// TwinCAT 3 PLC project PLC_MOTION
// Title: PLC_MOTION_LAYER
// Author: D. Hauer
// ProjectVersion: 01.01.00
// Description: MC-PtP, NCI, Camming cyclic execution layer for motion commands
// ProgramVersion: 3.1.4026.26
// CompilerDefines: TEST, NCI, CAM, XFC
// libraries:
//   Tc2_EtherCAT, * (Beckhoff Automation GmbH)
//   Tc2_MC2, * (Beckhoff Automation GmbH)
//   Tc2_MC2_Camming, * (Beckhoff Automation GmbH)
//   Tc2_MC2_Drive, * (Beckhoff Automation GmbH)
//   Tc2_MC2_FlyingSaw, * (Beckhoff Automation GmbH)
//   Tc2_MC2_XFC, * (Beckhoff Automation GmbH)
//   Tc2_NCI, * (Beckhoff Automation GmbH)
//   Tc2_PlcInterpolation, * (Beckhoff Automation GmbH)
//   Tc2_Standard, * (Beckhoff Automation GmbH)
//   Tc2_System, * (Beckhoff Automation GmbH)
//   Tc2_Utilities, * (Beckhoff Automation GmbH)
//   Tc3_Module, * (Beckhoff Automation GmbH)
// project tree:
//   APPLICATION/ GVL_APPLICATION.TcGVL (not stored)
//   APPLICATION/_types/Application/ E_APP_CHECK.TcDUT, E_APP_VARIANT.TcDUT (not stored), ST_APP_CTRL.TcDUT, ST_APP_STATE.TcDUT (not stored)
//   APPLICATION/_types/LinkedList/ E_LIST_CHECK.TcDUT, E_LIST_CTRL.TcDUT, E_LIST_STATE.TcDUT (not stored), fb_Process_LinkedList.TcPOU, fb_Process_LinkedListCtrl.TcPOU (not stored), I_Process_LinkedList.TcIO, ST_LIST_CTRL.TcDUT (not stored), ST_LIST_NODE_DATA.TcDUT (not stored), ST_LIST_STATE.TcDUT, ST_PROCESS_DATA.TcDUT (not stored), ST_PROCESS_LIST_RESULT.TcDUT
//   MAPPING/ MAPPING_AXIS_in.TcPOU, MAPPING_AXIS_out.TcPOU (not stored)
//   MAPPING/types/ U_AXIS_CTRL.TcDUT (not stored), U_AXIS_NC_PARAMETER_WRT.TcDUT, U_AXIS_HOMING.TcDUT (not stored), U_AXIS_MOTION_OPTIONS.TcDUT, U_AXIS_MOVE_DATA.TcDUT, U_AXIS_GEAR_IN.TcDUT (not stored), U_AXIS_NC_PARAMETER_RD.TcDUT, U_AXIS_STATE.TcDUT, U_AXIS_INFO.TcDUT (not stored), U_CAM_CTRL.TcDUT, U_CAM_DATA.TcDUT (not stored), U_CAM_INFO.TcDUT, U_CAM_STATE.TcDUT (not stored), U_FLY_CTRL.TcDUT (not stored), U_FLY_DATA.TcDUT, U_FLY_OPTIONS.TcDUT, U_FLY_STATE.TcDUT, U_NCI_AXIS_ID_GROUP.TcDUT, U_NCI_CTRL.TcDUT (not stored), U_NCI_INDEX_GROUP.TcDUT (not stored), U_NCI_R_PARAMETER_I.TcDUT (not stored), U_NCI_R_PARAMETER_Q.TcDUT (not stored), U_NCI_STATE.TcDUT (not stored), U_PARAMETER_SELECTOR_CTRL.TcDUT (not stored), U_PARAMETER_SELECTOR_STATE.TcDUT (not stored), U_TOUCH_PROBE_CTRL.TcDUT, U_TOUCH_PROBE_STATE.TcDUT, U_TRIGGER_CTRL.TcDUT, U_TRIGGER_STATE.TcDUT (not stored)
//   PLC_MOTION/CAM/ CAM.TcPOU, GVL_CAM.TcGVL (not stored)
//   PLC_MOTION/CAM/class/ FB_CamAxis.TcPOU, FB_CamCtrl.TcPOU (not stored), I_Cam_Ctrl.TcIO (not stored)
//   PLC_MOTION/CAM/types/ ST_CAM_CTRL.TcDUT (not stored), ST_CAM_DATA.TcDUT (not stored), ST_CAM_INFO.TcDUT (not stored), ST_CAM_OPTIONS.TcDUT (not stored), ST_CAM_READ_VALUES_PARAMETER.TcDUT (not stored), ST_CAM_SCALING_DATA.TcDUT (not stored), ST_CAM_STATE.TcDUT, ST_MOTION_FUNCTION.TcDUT (not stored), ST_MOTION_FUNCTION_POINT.TcDUT (not stored)
//   PLC_MOTION/FLYING_SAW/class/ FB_FlyingBase.TcPOU (not stored), FB_FlyingCtrl.TcPOU, I_Fly_Ctrl.TcIO
//   PLC_MOTION/FLYING_SAW/ FLYING_SAW.TcPOU (not stored), GVL_FLYING_SAW.TcGVL (not stored)
//   PLC_MOTION/FLYING_SAW/types/ ST_FLY_CTRL.TcDUT (not stored), ST_FLY_DATA.TcDUT (not stored), ST_FLY_OPTIONS.TcDUT, ST_FLY_STATE.TcDUT (not stored), ST_FLY_SYNC_MODE.TcDUT (not stored)
//   PLC_MOTION/FUNCTIONS/ FUNCTIONS.TcPOU (not stored), GVL_FUNCTIONS.TcGVL (not stored)
//   PLC_MOTION/FUNCTIONS/TOUCH_PROBE/ FB_TouchProbe.TcPOU, I_TouchProbe.TcIO (not stored)
//   PLC_MOTION/FUNCTIONS/TOUCH_PROBE/types/ ST_2BIT.TcDUT (not stored), ST_CTRL_TOUCH_PROBE.TcDUT, ST_DC_Input.TcDUT (not stored), ST_MTI_INPUT.TcDUT, ST_MTI_STATUS.TcDUT (not stored), ST_STATE_TOUCH_PROBE.TcDUT (not stored)
//   PLC_MOTION/FUNCTIONS/TRIGGER_BOX/ FB_TriggerBox.TcPOU (not stored), I_TriggerBox.TcIO (not stored)
//   PLC_MOTION/FUNCTIONS/TRIGGER_BOX/types/ ST_CTRL_TRIGGER.TcDUT (not stored), ST_DC_Output.TcDUT (not stored), ST_DC_State.TcDUT (not stored), ST_STATE_TRIGGER.TcDUT (not stored), T_TriggerControlBits.TcDUT (not stored)
//   PLC_MOTION/NCI/class/ FB_NciChannel.TcPOU (not stored), FB_NciChannelCtrl.TcPOU, I_NciChannel.TcIO (not stored), I_Nci_Ctrl.TcIO
//   PLC_MOTION/NCI/ GVL_NCI.TcGVL, NCI.TcPOU
//   PLC_MOTION/NCI/types/ E_NCI_CHANNEL_ERROR.TcDUT, E_NCI_CTRL.TcDUT, E_NCI_INTERPRETER_STATE.TcDUT, E_NCI_STATE.TcDUT, ST_3D_Group.TcDUT, ST_Index_Group.TcDUT (not stored), ST_Interface_Group.TcDUT, ST_NciChannel_Ref.TcDUT, ST_NCI_CTRL.TcDUT, ST_NCI_M_FUNC.TcDUT (not stored), ST_NCI_STATE.TcDUT, ST_R_Parameter.TcDUT (not stored)
//   PLC_MOTION/NC_PTP/class/ FB_McAxisBase.TcPOU (not stored), FB_McAxisCtrl.TcPOU, FB_ParameterSelector.TcPOU (not stored), I_McAxis.TcIO (not stored)
//   PLC_MOTION/NC_PTP/ GVL_AXIS.TcGVL (not stored), MAIN_AXIS.TcPOU
//   PLC_MOTION/NC_PTP/types/axis/ E_AxisEncoderType.TcDUT (not stored), ST_HomeParams.TcDUT (not stored)
//   PLC_MOTION/NC_PTP/types/control/ E_AXIS_CTRL.TcDUT (not stored), E_AXIS_SELECTOR.TcDUT, E_AXIS_STATE.TcDUT, ST_AXIS_CTRL.TcDUT, ST_AXIS_INFO.TcDUT (not stored), ST_AXIS_LIMIT_SWITCHES.TcDUT (not stored), ST_AXIS_STATE.TcDUT (not stored), ST_GEAR_IN.TcDUT (not stored), ST_HOMING.TcDUT (not stored), ST_MOTION_OPTIONS.TcDUT (not stored), ST_AXIS_MOVE_DATA.TcDUT (not stored), ST_NC_PARAMETER.TcDUT (not stored), ST_PARAMETER_SELECTOR_CTRL.TcDUT (not stored), ST_PARAMETER_SELECTOR_STATE.TcDUT
//   PLC_MOTION/XFC/ FB_Xfc.TcPOU
//   PLC_MOTION/XFC/types/ E_XFC_CHECK.TcDUT (not stored)
//   PLC_MOTION/_GVL/ GlobalTextList.TcGTLO, PLC_CONSTANT.TcGVL, PLC_VERSION.TcGVL
//   XTS_TRANSPORT/ GVL_XTS_CONSTANTS.TcGVL (not stored)
//   _MSG/class/ fb_LocalTime.TcPOU (not stored), fb_MessageData.TcPOU, fb_MessageDataCtrl.TcPOU (not stored)
//   _MSG/ GVL_MSG_XTS.TcGVL, f_MessageSet.TcPOU (not stored), GVL_MSG_AXIS.TcGVL, I_MessageData.TcIO
//   _types/ E_CHECK_STATE.TcDUT (not stored), E_PROGRESS.TcDUT (not stored), f_GetProgress.TcPOU (not stored), f_GetState.TcPOU (not stored), T_PROCESS.TcDUT (not stored)
//   _MSG/types/ e_Device.TcDUT, E_MessageType.TcDUT, E_MESSAGE_BATCH.TcDUT, E_MESSAGE_CHECK.TcDUT, E_MESSAGE_CTRL.TcDUT, E_MESSAGE_FLOW.TcDUT, E_MESSAGE_STATE.TcDUT, e_Subdevice.TcDUT, ST_Message.TcDUT, ST_MESSAGE_CTRL.TcDUT, ST_MESSAGE_STATE.TcDUT, TL_E_MESSAGETYPE.TcTLO
//   / PlcTask.TcTTO, Visualization Manager.TcVMO (not stored)
// (motion and I/O tree: see PLC project externcontrol)
// real-time tasks:
//   TASK PlcTask: cycle T#1ms, priority 20, ADS port 350
// variable links:
//   ExternControl/ExternControl Instance <-> PLC_MOTION/PLC_MOTION Instance
//     PlcTask Inputs/MAIN.eInitPlcMotion <-> PlcTask Outputs/MAIN_AXIS.eInit
//     PlcTask Inputs/MAPPING_in.AxisInfo.byState <-> PlcTask Outputs/MAPPING_AXIS_out.AxisInfo.byState
//     PlcTask Inputs/MAPPING_in.AxisParameterRd.byState <-> PlcTask Outputs/MAPPING_AXIS_out.AxisParameterOut.byState
//     PlcTask Inputs/MAPPING_in.AxisState.byState <-> PlcTask Outputs/MAPPING_AXIS_out.AxisState.byState
//     PlcTask Inputs/MAPPING_in.CamInfo.byState <-> PlcTask Outputs/MAPPING_AXIS_out.CamInfo.byState
//     PlcTask Inputs/MAPPING_in.CamState.byState <-> PlcTask Outputs/MAPPING_AXIS_out.CamState.byState
//     PlcTask Inputs/MAPPING_in.NciRparameters.byState <-> PlcTask Outputs/MAPPING_AXIS_out.NciRparameters.byCtrl
//     PlcTask Inputs/MAPPING_in.NciState.byState <-> PlcTask Outputs/MAPPING_AXIS_out.NciState.byState
//     PlcTask Inputs/MAPPING_in.TouchState.byState <-> PlcTask Outputs/MAPPING_AXIS_out.TouchProbeState.byState
//     PlcTask Inputs/MAPPING_in.TriggerState.byState <-> PlcTask Outputs/MAPPING_AXIS_out.TriggerState.byState
//     PlcTask Outputs/MAPPING_out.AxisCtrl.byCtrl <-> PlcTask Inputs/MAPPING_AXIS_in.AxisCtrl.byCtrl
//     PlcTask Outputs/MAPPING_out.AxisGearInData.byCtrl <-> PlcTask Inputs/MAPPING_AXIS_in.AxisGearInData.byCtrl
//     PlcTask Outputs/MAPPING_out.AxisHoming.byCtrl <-> PlcTask Inputs/MAPPING_AXIS_in.AxisHoming.byCtrl
//     PlcTask Outputs/MAPPING_out.AxisMotionOptions.byCtrl <-> PlcTask Inputs/MAPPING_AXIS_in.AxisMotionOptions.byCtrl
//     PlcTask Outputs/MAPPING_out.AxisMoveData.byCtrl <-> PlcTask Inputs/MAPPING_AXIS_in.AxisMoveData.byCtrl
//     PlcTask Outputs/MAPPING_out.AxisParameterWrt.byCtrl <-> PlcTask Inputs/MAPPING_AXIS_in.AxisParameterIn.byCtrl
//     PlcTask Outputs/MAPPING_out.CamCtrl.byCtrl <-> PlcTask Inputs/MAPPING_AXIS_in.CamControl.byCtrl
//     PlcTask Outputs/MAPPING_out.CamData.byCtrl <-> PlcTask Inputs/MAPPING_AXIS_in.CamData.byCtrl
//     PlcTask Outputs/MAPPING_out.NciAxisGroup.byCtrl <-> PlcTask Inputs/MAPPING_AXIS_in.NciAxisGroup.byCtrl
//     PlcTask Outputs/MAPPING_out.NciControl.byCtrl <-> PlcTask Inputs/MAPPING_AXIS_in.NciControl.byCtrl[1]
//     PlcTask Outputs/MAPPING_out.NciRparameters.byCtrl <-> PlcTask Inputs/MAPPING_AXIS_in.NciRparameters.byCtrl
//     PlcTask Outputs/MAPPING_out.TouchCtrl.byCtrl <-> PlcTask Inputs/MAPPING_AXIS_in.TouchProbeControl.byCtrl
//     PlcTask Outputs/MAPPING_out.TriggerCtrl.byCtrl <-> PlcTask Inputs/MAPPING_AXIS_in.TriggerControl.byCtrl
//   PLC_MOTION/PLC_MOTION Instance <-> NC-Task 1 SAF/Axes/Axis 6
//     PlcTask Inputs/GVL_AXIS.AxisRef[6].NcToPlc <-> Outputs/ToPlc
//     PlcTask Outputs/GVL_AXIS.AxisRef[6].PlcToNc <-> Inputs/FromPlc
//   PLC_MOTION/PLC_MOTION Instance <-> NC-Task 1 SAF/Axes/AxisX
//     PlcTask Inputs/GVL_AXIS.AxisRef[1].NcToPlc <-> Outputs/ToPlc
//     PlcTask Outputs/GVL_AXIS.AxisRef[1].PlcToNc <-> Inputs/FromPlc
//   PLC_MOTION/PLC_MOTION Instance <-> NC-Task 1 SAF/Axes/AxisY
//     PlcTask Inputs/GVL_AXIS.AxisRef[2].NcToPlc <-> Outputs/ToPlc
//     PlcTask Outputs/GVL_AXIS.AxisRef[2].PlcToNc <-> Inputs/FromPlc
//   PLC_MOTION/PLC_MOTION Instance <-> NC-Task 1 SAF/Axes/AxisZ
//     PlcTask Inputs/GVL_AXIS.AxisRef[3].NcToPlc <-> Outputs/ToPlc
//     PlcTask Outputs/GVL_AXIS.AxisRef[3].PlcToNc <-> Inputs/FromPlc
//   PLC_MOTION/PLC_MOTION Instance <-> NC-Task 1 SAF/Axes/Dos_A1
//     PlcTask Inputs/GVL_AXIS.AxisRef[4].NcToPlc <-> Outputs/ToPlc
//     PlcTask Outputs/GVL_AXIS.AxisRef[4].PlcToNc <-> Inputs/FromPlc
//   PLC_MOTION/PLC_MOTION Instance <-> NC-Task 1 SAF/Axes/Dos_A2
//     PlcTask Inputs/GVL_AXIS.AxisRef[5].NcToPlc <-> Outputs/ToPlc
//     PlcTask Outputs/GVL_AXIS.AxisRef[5].PlcToNc <-> Inputs/FromPlc
//   PLC_MOTION/PLC_MOTION Instance <-> NC-Task 1 SAF/Channel XYZ
//     PlcTask Inputs/GVL_NCI.NciCtrl[1]._stChannelRef.NcToPlc <-> Outputs/ToPlc
//     PlcTask Outputs/GVL_NCI.NciCtrl[1]._stChannelRef.PlcToNc <-> Inputs/FromPlc

CONFIGURATION PLC_MOTION
    RESOURCE PLC ON TwinCAT3
        TASK PlcTask(INTERVAL := T#1ms, PRIORITY := 20);
        PROGRAM MAPPING_AXIS_in WITH PlcTask : MAPPING_AXIS_in;
        PROGRAM MAIN_AXIS WITH PlcTask : MAIN_AXIS;
        PROGRAM FUNCTIONS WITH PlcTask : FUNCTIONS;
        PROGRAM NCI WITH PlcTask : NCI;
        PROGRAM CAM WITH PlcTask : CAM;
        PROGRAM FLYING_SAW WITH PlcTask : FLYING_SAW;
        PROGRAM MAPPING_AXIS_out WITH PlcTask : MAPPING_AXIS_out;
    END_RESOURCE
END_CONFIGURATION

// ---- APPLICATION/_types/Application/E_APP_CHECK.TcDUT
{attribute 'qualified_only'}
{attribute 'strict'}
{attribute 'to_string'}
TYPE E_APP_CHECK :
(
  NULL,

  POINTER_CTRL_INVALID                := 9000,
  POINTER_STATE_INVALID,
  REFERENCE_INSTANCE_CONTROL_INVALID,
  REFERENCE_INSTANCE_STATE_INVALID,

	POINTER_TRANSPORT_CTRL_INVALID      := 9100,
	POINTER_TRANSPORT_STATE_INVALID     := 9200,
	POINTER_COLLECTOR_ITF_INVALID       := 9300,
  REFERENCE_PROCESS_LIST_ITF_INVALID  := 9400,

  CHECK_DONE := 10000

)UINT;
END_TYPE

// ---- APPLICATION/_types/Application/ST_APP_CTRL.TcDUT
TYPE ST_APP_CTRL :
STRUCT
  Cmd       : E_INSTANCE_CMD;
  Variant   : E_APP_VARIANT;
END_STRUCT
END_TYPE

// ---- APPLICATION/_types/LinkedList/E_LIST_CHECK.TcDUT
{attribute 'qualified_only'}
{attribute 'strict'}
{attribute 'to_string'}
TYPE E_LIST_CHECK :
(
	NULL,
  REFERENCE_CTRL_INVALID := 9000,
  REFERENCE_STATE_INVALID,
  REFERENCE_DATA_INPUT_INVALID,
  REFERENCE_DATA_OUTPUT_INVALID,

  CHECK_DONE              := 10000
);
END_TYPE

// ---- APPLICATION/_types/LinkedList/E_LIST_CTRL.TcDUT
{attribute 'qualified_only'}
{attribute 'strict'}
{attribute 'to_string'}
TYPE E_LIST_CTRL :
(
  LIST_CTRL_INVALID,
	LIST_CTRL_NULL,
  LIST_CTRL_INIT      := 10,
  LIST_CTRL_GET_HEAD  := 20,
  LIST_CTRL_GET_TAIL  := 30,
  LIST_CTRL_ADD_HEAD  := 40,
  LIST_CTRL_ADD_TAIL  := 50,
  LIST_CTRL_DEL_HEAD  := 60,
  LIST_CTRL_DEL_TAIL  := 70
)UINT;
END_TYPE

// ---- APPLICATION/_types/LinkedList/ST_LIST_STATE.TcDUT
{attribute 'pack_mode' := '2'}
TYPE ST_LIST_STATE :
STRUCT
  Init        : E_PROGRESS;
  State       : E_LIST_STATE;

  Free        : UDINT;
  Count       : UDINT;
END_STRUCT
END_TYPE

// ---- APPLICATION/_types/LinkedList/ST_PROCESS_LIST_RESULT.TcDUT
TYPE ST_PROCESS_LIST_RESULT :
STRUCT
  wState    : WORD;   // wState == 0 --> all ok
  nIndex    : ULINT;
  stData    : ST_PROCESS_DATA;  // copy of list entry
END_STRUCT
END_TYPE

// ---- MAPPING/types/U_AXIS_NC_PARAMETER_WRT.TcDUT
TYPE U_AXIS_NC_PARAMETER_WRT :
UNION

  stCtrl              : ARRAY[1..MAX_AXIS] OF ST_NC_PARAMETER;

  byCtrl    AT %I*    : ARRAY[1..MAX_AXIS] OF
                        ARRAY[1..SIZEOF(ST_NC_PARAMETER)] OF BYTE;
END_UNION
END_TYPE

// ---- MAPPING/types/U_AXIS_MOTION_OPTIONS.TcDUT
TYPE U_AXIS_MOTION_OPTIONS :
UNION

  stCtrl              : ARRAY[1..MAX_AXIS] OF ST_MOTION_OPTIONS;

  byCtrl    AT %I*    : ARRAY[1..MAX_AXIS] OF
                        ARRAY[1..SIZEOF(ST_MOTION_OPTIONS)] OF BYTE;
END_UNION
END_TYPE

// ---- MAPPING/types/U_AXIS_MOVE_DATA.TcDUT
TYPE U_AXIS_MOVE_DATA :
UNION

  stCtrl              : ARRAY[1..MAX_AXIS] OF ST_AXIS_MOVE_DATA;

  byCtrl    AT %I*    : ARRAY[1..MAX_AXIS] OF
                        ARRAY[1..SIZEOF(ST_AXIS_MOVE_DATA)] OF BYTE;
END_UNION
END_TYPE

// ---- MAPPING/types/U_AXIS_NC_PARAMETER_RD.TcDUT
TYPE U_AXIS_NC_PARAMETER_RD :
UNION

  stState             : ARRAY[1..MAX_AXIS] OF ST_NC_PARAMETER;

  byState   AT %Q*    : ARRAY[1..MAX_AXIS] OF
                        ARRAY[1..SIZEOF(ST_NC_PARAMETER)] OF BYTE;
END_UNION
END_TYPE

// ---- MAPPING/types/U_AXIS_STATE.TcDUT
TYPE U_AXIS_STATE :
UNION

  stState             : ARRAY[1..MAX_AXIS] OF ST_AXIS_STATE;

  byState   AT %Q*    : ARRAY[1..MAX_AXIS] OF
                        ARRAY[1..SIZEOF(ST_AXIS_STATE)] OF BYTE;
END_UNION
END_TYPE

// ---- MAPPING/types/U_CAM_CTRL.TcDUT
TYPE U_CAM_CTRL :
UNION
  stCtrl              : ARRAY[1..MAX_AXIS] OF ST_CAM_CTRL;

  byCtrl    AT %I*    : ARRAY[1..MAX_AXIS] OF
                        ARRAY[1..SIZEOF(ST_CAM_CTRL)] OF BYTE;
END_UNION
END_TYPE

// ---- MAPPING/types/U_CAM_INFO.TcDUT
TYPE U_CAM_INFO :
UNION

  stState             : ARRAY[1..MAX_AXIS] OF ST_CAM_INFO;

  byState  AT %Q*     : ARRAY[1..MAX_AXIS] OF
                        ARRAY[1..SIZEOF(ST_CAM_INFO)] OF BYTE;
END_UNION
END_TYPE

// ---- MAPPING/types/U_FLY_DATA.TcDUT
TYPE U_FLY_DATA :
UNION

  stCtrl              : ARRAY[1..MAX_AXIS] OF ST_FLY_DATA;

  byCtrl    AT %I*    : ARRAY[1..MAX_AXIS] OF
                        ARRAY[1..SIZEOF(ST_FLY_DATA)] OF BYTE;

END_UNION
END_TYPE

// ---- MAPPING/types/U_FLY_OPTIONS.TcDUT
TYPE U_FLY_OPTIONS :
UNION

  stCtrl              : ARRAY[1..MAX_AXIS] OF ST_FLY_OPTIONS;

  byCtrl    AT %I*    : ARRAY[1..MAX_AXIS] OF
                        ARRAY[1..SIZEOF(ST_FLY_OPTIONS)] OF BYTE;

END_UNION
END_TYPE

// ---- MAPPING/types/U_FLY_STATE.TcDUT
TYPE U_FLY_STATE :
UNION

  stState             : ARRAY[1..MAX_AXIS] OF ST_FLY_STATE;

  byState   AT %Q*    : ARRAY[1..MAX_AXIS] OF
                        ARRAY[1..SIZEOF(ST_FLY_STATE)] OF BYTE;
END_UNION
END_TYPE

// ---- MAPPING/types/U_NCI_AXIS_ID_GROUP.TcDUT
TYPE U_NCI_AXIS_ID_GROUP :
UNION

  stCtrl              : ARRAY[1..MAX_NCI_CH] OF ST_3D_Group;

  byCtrl    AT %I*    : ARRAY[1..MAX_NCI_CH] OF
                        ARRAY[1..SIZEOF(ST_3D_Group)] OF BYTE;
END_UNION
END_TYPE

// ---- MAPPING/types/U_TOUCH_PROBE_CTRL.TcDUT
TYPE U_TOUCH_PROBE_CTRL :
UNION
  stCtrl              : ARRAY[1..MAX_TOUCH_PROBE] OF ST_CTRL_TOUCH_PROBE;

  byCtrl    AT %I*    : ARRAY[1..MAX_TOUCH_PROBE] OF
                        ARRAY[1..SIZEOF(ST_CTRL_TOUCH_PROBE)] OF BYTE;
END_UNION
END_TYPE

// ---- MAPPING/types/U_TOUCH_PROBE_STATE.TcDUT
TYPE U_TOUCH_PROBE_STATE :
UNION
  stState              : ARRAY[1..MAX_TOUCH_PROBE] OF ST_STATE_TOUCH_PROBE;

  byState    AT %Q*   : ARRAY[1..MAX_TOUCH_PROBE] OF
                        ARRAY[1..SIZEOF(ST_STATE_TOUCH_PROBE)] OF BYTE;
END_UNION
END_TYPE

// ---- MAPPING/types/U_TRIGGER_CTRL.TcDUT
TYPE U_TRIGGER_CTRL :
UNION
  stCtrl              : ARRAY[1..MAX_TRIGGER_BOX] OF ST_CTRL_TRIGGER;

  byCtrl    AT %I*    : ARRAY[1..MAX_TRIGGER_BOX] OF
                        ARRAY[1..SIZEOF(ST_CTRL_TRIGGER)] OF BYTE;
END_UNION
END_TYPE

// ---- PLC_MOTION/CAM/types/ST_CAM_STATE.TcDUT
{attribute 'pack_mode' := '2'}
TYPE ST_CAM_STATE :
STRUCT
  bError              : BIT;

  eState              : E_AXIS_STATE; // mirror the requested command + E_PROGRESS

  wCamCouplingState   : ARRAY[0..7] OF WORD;
  nCamCouplingTableId : ARRAY[0..7] OF UINT;

  nNumPointsRead      : UDINT;
END_STRUCT
END_TYPE

// ---- PLC_MOTION/FLYING_SAW/types/ST_FLY_OPTIONS.TcDUT
{attribute 'pack_mode' := '2'}
TYPE ST_FLY_OPTIONS :
STRUCT
  PositionLimitMin        : LREAL ; // will additionally be checked if GearInSync_CheckMask_OptionalMinPos is set to TRUE  
  PositionLimitMax        : LREAL ; // will additionally be checked if GearInSync_CheckMask_OptionalMaxPos is set to TRUE

  SyncMode                : ST_FLY_SYNC_MODE;
END_STRUCT
END_TYPE

// ---- PLC_MOTION/FUNCTIONS/TOUCH_PROBE/types/ST_CTRL_TOUCH_PROBE.TcDUT
TYPE ST_CTRL_TOUCH_PROBE :
STRUCT
  Enable        : BIT;

  AxisId        : UDINT;      // TwinCAT NC Axis ID

  SensorIndex   : UDINT;      // sensor select; 1 := upper , 2 := lower, 0 := default upper 

  Direction     : INT := 1;   // typeof(MC_DIRECTION)
                                // MC_Positive_Direction := 1,   -(set trigger when crossing moving in pos dir)
                                // MC_Shortest_Way,               (not used in TouchProbe or TriggerBox)
                                // MC_Negative_Direction := 3,   -(set trigger when crossing moving in neg dir)
                                // MC_Current_Direction  := 4,    (not used in TouchProbe or TriggerBox)
                                // MC_Undefined_Direction := 128  (not used in TouchProbe or TriggerBox)

  PositionStart : LREAL; // axis has to reach this position in order to start the check for change in input timestamp
  PositionEnd   : LREAL; // axis must not reach this position without state change on input --> error
END_STRUCT
END_TYPE

// ---- PLC_MOTION/FUNCTIONS/TOUCH_PROBE/types/ST_MTI_INPUT.TcDUT
TYPE ST_MTI_INPUT :
STRUCT
  EventState            : BIT;
  EventTime             : UDINT;
END_STRUCT
END_TYPE

// ---- PLC_MOTION/NCI/types/E_NCI_CHANNEL_ERROR.TcDUT
{attribute 'qualified_only'}
{attribute 'strict'}
TYPE E_NCI_CHANNEL_ERROR :
(
  e_Null,
  e_InvalidReference_ChannelRef,
  e_AxisConfigurationMismatch_McAxis,
  e_AxisConfigurationMismatch_AuxAxis


);
END_TYPE

// ---- PLC_MOTION/NCI/types/E_NCI_CTRL.TcDUT
{attribute 'qualified_only'}
{attribute 'strict'}
{attribute 'to_string'}
TYPE E_NCI_CTRL :
(
  NULL,
  INIT,
  IDLE,
  RESET,
  LOAD_PROG,
  FEED_TABLE,
  BUILD_GROUP,
  CLEAR_GROUP,

  START         := 10,
  STOP,
  STO_STOP,
  RESTART_STEP_ON,

  M_FUNC_QUIT   := 20,

  READ_R_PARA   := 30,
  WRITE_R_PARA  := 40

)UINT;
END_TYPE

// ---- PLC_MOTION/NCI/types/E_NCI_INTERPRETER_STATE.TcDUT
// Interpreter state, see also library tc2_nci.Global_Variables.NCI_INTERPRETER_xxx
//  Date    Name  Version   Remarks
//  2016/09/29  FJK   1.0     1st Version
{attribute -'to_string'}
TYPE E_NCI_INTERPRETER_STATE :
(
  NCI_INTERPRETER_INITFAILED := 0,
  NCI_INTERPRETER_IDLE := 1,
  NCI_INTERPRETER_READY := 2,
  NCI_INTERPRETER_STARTED := 3,
  NCI_INTERPRETER_SCANNING := 4,
  NCI_INTERPRETER_RUNNING := 5,
  NCI_INTERPRETER_STAY_RUNNING := 6,
  NCI_INTERPRETER_WRITETABLE := 7,
  NCI_INTERPRETER_SEARCHLINE := 8,
  NCI_INTERPRETER_END := 9,
  NCI_INTERPRETER_SINGLESTOP := 10, 
  NCI_INTERPRETER_ABORTING := 11,
  NCI_INTERPRETER_ABORTED := 12,
  NCI_INTERPRETER_FAULT := 13,
  NCI_INTERPRETER_RESET := 14,
  NCI_INTERPRETER_STOP := 15,
  NCI_INTERPRETER_WAITFUNC := 16,
  NCI_INTERPRETER_FLUSHBUFFERS := 17
) DWORD;    //Basis-Datentyp
END_TYPE

// ---- PLC_MOTION/NCI/types/E_NCI_STATE.TcDUT
{attribute 'qualified_only'}
//{attribute 'strict'}
{attribute 'to_string'}
TYPE E_NCI_STATE :
(
  NULL,
  INIT,
  IDLE,
  RESET,
  LOAD_PROG,
  FEED_TABLE,
  BUILD_GROUP,
  CLEAR_GROUP,

  START         := 10,
  STOP,
  STO_STOP,
  RESTART_STEP_ON,

  M_FUNC_QUIT   := 20,

  READ_R_PARA   := 30,
  WRITE_R_PARA  := 40

)UINT;
END_TYPE

// ---- PLC_MOTION/NCI/types/ST_3D_Group.TcDUT
{attribute 'pack_mode' := '2'}
TYPE ST_3D_Group :
STRUCT
  nXAxisId    : UDINT := 1;
  nYAxisId    : UDINT := 2;
  nZAxisId    : UDINT := 3;
  nQ1AxisId   : UDINT;
  nQ2AxisId   : UDINT;
  nQ3AxisId   : UDINT;
  nQ4AxisId   : UDINT;
  nQ5AxisId   : UDINT;
END_STRUCT
END_TYPE

// ---- PLC_MOTION/NCI/types/ST_Interface_Group.TcDUT
{attribute 'pack_mode' := '2'}
TYPE ST_Interface_Group :
STRUCT
  I_Idx_XAxis     : I_McAxis;
  I_Idx_YAxis     : I_McAxis;
  I_Idx_ZAxis     : I_McAxis;

  I_Idx_Q1Axis    : I_McAxis;
  I_Idx_Q2Axis    : I_McAxis;
  I_Idx_Q3Axis    : I_McAxis;
  I_Idx_Q4Axis    : I_McAxis;
  I_Idx_Q5Axis    : I_McAxis;
END_STRUCT
END_TYPE

// ---- PLC_MOTION/NCI/types/ST_NciChannel_Ref.TcDUT
TYPE ST_NciChannel_Ref :
STRUCT
  NcToPlc AT %I*: NcToPlc_NciChannel_Ref;   //  Externer Datentyp!
  PlcToNc AT %Q*: PlcToNc_NciChannel_Ref;   //  Externer Datentyp!
END_STRUCT
END_TYPE

// ---- PLC_MOTION/NCI/types/ST_NCI_CTRL.TcDUT
{attribute 'pack_mode' := '2'}
TYPE ST_NCI_CTRL :
STRUCT
  eCmd          : E_NCI_CTRL := E_NCI_CTRL.INIT;
  rOverride     : REAL := 47.11;

  sProgramName  : STRING(255);
END_STRUCT
END_TYPE

// ---- PLC_MOTION/NCI/types/ST_NCI_STATE.TcDUT
{attribute 'pack_mode' := '2'}
TYPE ST_NCI_STATE :
STRUCT
  eState        : E_NCI_STATE; // eCmd with offsets E_PROGRESS

  bMFuncReq     : BIT;  // M function request is active from channel

  nMFunc        : WORD; // number of active M function

  nItpState     : UINT; 
                         (*  Interpreter Operation State:
                            0  = Init failed
                            1  = Idle
                            2  = Ready
                            3  = Started
                            4  = Scanning
                            5  = Running
                            6  = Stay running
                            7  = Write table
                            8  = Search line
                            9  = End
                            10 = Single Step
                            11 = Aborting
                            12 = Aborted
                            13 = Fault
                            14 = Reset
                            15 = Stop
                            16 = Wait function
                            17 = Flush buffers
                          *) 

  rAxisOverride       : LREAL; // active override in cyclic NCI interface
  sProgramNameActive  : STRING(255);
END_STRUCT
END_TYPE

// ---- PLC_MOTION/NC_PTP/types/control/E_AXIS_SELECTOR.TcDUT
{attribute 'qualified_only'}
{attribute 'strict'}
{attribute 'to_string'}
TYPE E_AXIS_SELECTOR :
(
	SELECT_INDEX,
  SELECT_AXIS_ID
);
END_TYPE

// ---- PLC_MOTION/NC_PTP/types/control/E_AXIS_STATE.TcDUT
{attribute 'qualified_only'}
{attribute 'to_string'}
TYPE E_AXIS_STATE :
(
  AXIS_NULL,   // null reaction to command
  AXIS_INIT,
  AXIS_DISABLE,
  AXIS_ENABLE,

  AXIS_NO_INIT  := 9,
  
  AXIS_IDLE     := 10, // clear axis and enable
  AXIS_HOME,
  AXIS_MOVE_POS,
  AXIS_MOVE_VELO,
  AXIS_HALT,
  AXIS_STOP,
  AXIS_SEND_TO_POS,

  AXIS_RESET              := 19,
  AXIS_STARTUP            := 20,

  AXIS_MOVE_BUFFER        := 30,
  AXIS_MOVE_BUFFER_VELO,

  AXIS_PARAMETER_READ     := 40, // command for reading and writing parameter
  AXIS_PARAMETER_WRITE,
  AXIS_PARAMETER_WRITE_PERSISTENT,


  AXIS_GEAR_IN            := 50,
  AXIS_GEAR_OUT,
  AXIS_GEAR_IN_MULTIMASTER,

  CAM_INIT                := 60,
  CAM_IN,
  CAM_OUT,
  CAM_SCALING,
  CAM_INFO,
  CAM_RD_MOTION_FUNCTION,
  CAM_RD_MOTION_FUNCTION_POINT,
  CAM_RD_MOTION_FUNCTIONS_VALUES,
  CAM_WRT_MOTION_FUNCTION,
  CAM_WRT_MOTION_FUNCTION_POINT,

  FLY_GEAR_IN_POS         := 70,
  FLY_GEAR_IN_VELO

)UINT;
END_TYPE

// ---- PLC_MOTION/NC_PTP/types/control/ST_AXIS_CTRL.TcDUT
{attribute 'pack_mode' := '2'}
TYPE ST_AXIS_CTRL :
STRUCT
  eCmd                : E_AXIS_CTRL;    // commanded axis function
  eProgress           : E_PROGRESS;     // progress command for synced functions
END_STRUCT
END_TYPE

// ---- PLC_MOTION/NC_PTP/types/control/ST_PARAMETER_SELECTOR_STATE.TcDUT
TYPE ST_PARAMETER_SELECTOR_STATE :
STRUCT
  AxisIndex   : UINT;             // what you selected mirrored back
  AxisId      : UDINT;            // matching Id to the index
  State       : ST_AXIS_STATE;    // result identifier to your command
  Info        : ST_NC_PARAMETER;  // read data
END_STRUCT
END_TYPE

// ---- _MSG/types/e_Device.TcDUT
{attribute 'to_string'}
TYPE e_Device :
(
  // txt file logging LOG_FILE
  Device_Null,                  // NULL               - not to be used
  Device_Main,                  // MAIN(PRG)          - reserved for MAIN(PRG)
  Device_MainAxis,              // MAIN_AXIS(PRG)     - reserved for MAIN_AXIS(PRG)
  Device_Nci,                   // NCI(PRG)           - reserved for NCI(PRG)
  Device_Cam,                   // CAM(PRG            - reserved for CAM(PRG)
  Device_Functions,             // FUNCTIONS(PRG)     - reserved for FUNCTIONS(PRG)
  Device_FlyingSaw,             // FLYING_SAW(PRG)    - reserved for FLYING_SAW(PRG)
  Device_MainApplication,       // MAIN_APP(PRG)

  Device_MoverSelector,         // single mover interface for xts applications
  Device_ParameterSelector,     // fb_ParameterSelector can only exist once in a project.
  Device_Configuration,         // fb_Configuration can handle multiple files therefore only one instance is required
  Device_XmlData,               // generic XML Data (e.g. persistent data)
  Device_Utilities,             // service calls to anyone you may want to talk to, the main intent is to get XPU and TcXtsIo data to the application side


  General           :=  1000,
  CaGroup           :=  2000,
  Xpu               :=  3000,
  XpuCtrl           :=  4000,
  Mover             :=  5000,
  MoverCtrl         :=  6000,
  XtsTransportUnit  :=  7000,
  XfcTriggerBox     :=  8000,
  XfcTouchProbe     :=  9000,
  XtsStation        := 10000,

  Camming           := 11000,
  NciChannel        := 12000,
  NciChannelCtrl    := 13000,
  Axis              := 14000,
  XfcAxis           := 15000,

  // txt file logging LOG_FILE_METRICS
  MetricsXts        := 16000,   //entries from xts Metrics are written into dedicated txt file (see f_MessageSet, here's the diverter)
  MetricsAxis       := 17000,   //entries from PLC_MOTION Metrics are written into dedicated txt file

  FlyingSaw         := 18000,


  // txt file logging LOG_FILE_APP
  Process           := 20000,
  ProcessListCtrl   := 21000,
  TicketListCtrl    := 22000,

  Application       := 30000,

  // txt file logging LOG_FILE_PRODUCT - this is for you to use
  DataProduct       := 40000
)UDINT;
END_TYPE

// ---- _MSG/types/E_MessageType.TcDUT
{attribute 'strict'}
{attribute 'to_string'}
TYPE E_MessageType :
(
  //-----------------------------------------------------
  //-----------------------------------------------------
  //  message system:
  //  - errors are always calling f_MessageSet()
  //  - errors are always entered into its list
  //
  //  - message severity is set by this enum (like everywhere else)
  //
  //  - message frequency is set by this enum
  //    - IF you get above 50 stations, 
  //      writing to the file system takes time:
  //
  //    Batch: switching on metrics (> Empty) must not add cpu load, 
  //      --> so do not clutter here
  //
  //    Info:  regular flow of information (>Error / >Warning) 
  //           must not add significant cpu load, 
  //      --> so do not clutter here
  //
  //    Verbose and above:
  //    --> for small systems (< 96 mover, < 50 stations) 
  //        you may switch it on for everybody, 
  //        files get big quickly ;-)
  //
  //    --> switch on during test phase for a handful of stations
  //
  //    --> high detail logging always and for everybody
  //    --> we need somebody who transfers data more quickly
  //      --> I can offer a .NET(C#) ADS tool which collects the list.
  //          .NET application then pushes to database
  //-----------------------------------------------------
  //-----------------------------------------------------
  eMessageEmpty,    // he who is without bounds may speak
  eMessageBatch,    // he who counts words, counts numbers (Batch started, Next in Batch, Batch done)
  eMessageError,    // mine, your(')s, anybody's, let the numbers tell you
  eMessageWarning,  // I told you so
  eMessageInfo,     // A long time ago in a galaxy far, far away...
  eMessageVerbose,  // He talks a lot, doesn't he?; Yeah! He's very knowledgeable.
  eMessageSentient  // Keep them out of bright light, Don't get them wet, do not feed them after midnight!! No matter how much they beg!!
)DINT;
END_TYPE

// ---- _MSG/types/E_MESSAGE_BATCH.TcDUT
{attribute 'qualified_only'}
{attribute 'strict'}
{attribute 'to_string'}
TYPE E_MESSAGE_BATCH :
(
	MSG_BATCH_NULL,
  MSG_BATCH_JOB_STARTED,
  MSG_BATCH_NEXT_IN_JOB,
  MSG_BATCH_JOB_DONE
)UINT;
END_TYPE

// ---- _MSG/types/E_MESSAGE_CHECK.TcDUT
{attribute 'qualified_only'}
{attribute 'strict'}
{attribute 'to_string'}
TYPE E_MESSAGE_CHECK :
(
  // 9000 --> here comes your error
  MSG_CHECK_INVALID_POINTER             := 9000,
  MSG_CHECK_INVALID_POINTER_TIME,
  MSG_CHECK_INVALID_POINTER_LIST,
  MSG_CHECK_INVALID_POINTER_MSG_IDX,
  MSG_CHECK_INVALID_POINTER_ERR_IDX,
  MSG_CHECK_INVALID_POINTER_ROOT_FILE,
  MSG_CHECK_INVALID_POINTER_ROOT_DIR,
  MSG_CHECK_INVALID_POINTER_CTRL,
  MSG_CHECK_INVALID_POINTER_STATE,

  // 10000 --> here comes your man
  MSG_CHECK_DONE                        := 10000
)UINT;
END_TYPE

// ---- _MSG/types/E_MESSAGE_CTRL.TcDUT
{attribute 'qualified_only'}
{attribute 'strict'}
{attribute 'to_string'}
TYPE E_MESSAGE_CTRL :
(
	MSG_CTRL_NULL,
	MSG_CTRL_INIT   := 10,
  MSG_CTRL_IDLE   := 30,
  MSG_CTRL_WRITE  := 50
)UINT;
END_TYPE

// ---- _MSG/types/E_MESSAGE_FLOW.TcDUT
{attribute 'qualified_only'}
{attribute 'strict'}
{attribute 'to_string'}
TYPE E_MESSAGE_FLOW :
(
  MSG_FLOW_INIT,
  MSG_FLOW_ROOT                 := 10,
  MSG_FLOW_ROOT_CREATE,
  MSG_FLOW_ROOT_CREATE_BUSY,
  MSG_FLOW_FOLDER,
  MSG_FLOW_FOLDER_CREATE,
  MSG_FLOW_FOLDER_CREATE_BUSY,
  MSG_FLOW_FILE_CREATE_DONE,
  MSG_FLOW_LINE_START           := 100,
  MSG_FLOW_LINE_BUILD,
  MSG_FLOW_LINE_CHECK,
  MSG_FLOW_WRITE_FILE_BUSY      := 200,
  MSG_FLOW_WRITE_FILE_END,
  MSG_FLOW_WRITE_FILE_DONE      := 1000
)UINT;
END_TYPE

// ---- _MSG/types/E_MESSAGE_STATE.TcDUT
{attribute 'qualified_only'}
//{attribute 'strict'}
{attribute 'to_string'}
TYPE E_MESSAGE_STATE :
(
	MSG_STATE_NULL,
  MSG_STATE_INIT    := 10,
  MSG_STATE_IDLE    := 30,
  MSG_STATE_WRITE   := 50
)UINT;
END_TYPE

// ---- _MSG/types/e_Subdevice.TcDUT
{attribute 'strict'}
{attribute 'to_string'}
TYPE e_Subdevice :
(
  // sub device for message system
  General                 :=  0,
  MainInit,
  // Motion Control FB Instances
  fbPower,
  fbReset,
  fbResetSercos,
  fbHalt,
  fbStop,                 // 5
  fbHome,
  fbJog,
  fbMoveVelocity1,
  fbMoveVelocity2,
  fbMoveAbsolute1,        // 10
  fbMoveAbsolute2,
  fbMoveEndless,
  fbMovePtP,
  fbMoveVelo,

  // CA CollisionAvoidance FB instances
  // CA group fb instances
  fbCaGroup             := 30,
  fbMoveToPosCa,
  fbSendToAbsPosCa,
  fbSendToModuloPosCa,
  fbGearInPosCa,
  fbGroupAddAxis,
  fbGroupRemoveAxis,
  fbGroupDisable,
  fbGroupEnable,
  fbGroupErrorRead,
  fbGroupStatusRead,
  fbGroupReset,
  fbGroupStop,
  fbHaltCa,
  fbSendToPos,

  fbGearIn                := 50,
  fbGearOut,
  fbGearInMultiMaster,

  fbGearInPos,
  fbGearInVelo,


  fbCamOut                := 80,
  fbCamInV2,
  fbCamScalingV2,
  fbCamInfoV2,
  fbReadMotionFunction,
  fbReadMotionFunctionPoint,
  fbReadMotionFunctionValues,
  fbWriteMotionFunction,
  fbWriteMotionFunctionPoint,
  fbSetOnlineChangeMode,

  fbReadParameter         := 100,
  fbReadBoolParameter,
  fbWriteParameter,
  fbWriteBoolParameter,
  fbWriteParameterPersistent,

  fbBuildGroup            := 200,
  fbClearGroup,
  fbLoadProg,
  fbResetItp,
  fbStartStopItp,
  fbEStopItp,             // 205
  fbStepOnAfterEStopItp,
  fbConfirmHskItp,
  fbDelDtgItp,
  fbNciFeedTablePreparation,
  fbNciFeedTable,         // 210
  fbReadLine,
  fbItpReadRParams,
  fbItpWriteRParams,
  Get_ItpState,
  Get_Error,              // 215


  XfcPositionAtTime       := 300,
  XfcTimeOfPosition,
  XfcTimeToPosition,
  XfcTimeToModuloPosition,
  XfcRecordedPosition,
  XfcTouchProbe,          // 305
  XfcTouchProbeEL1258,
  XfcTouchProbeOptions,
  XfcTriggerRef,
  XfcTriggerRef_MT,
  XfcEl1258Interface_MT,  // 310
  XfcRecordedPosition_MT,
  XfcTriggerOut,
  XfcTriggerStart,
  XfcSwitchOn_2252,
  XfcSwitchOff_2252,      // 315
  XfcInit,
  XfcLatchPosition,
  XfcWaitForPosition,

  AxisMode              := 1000,
  AxisControl,
  AxisStartUp,
  AxisCycle,
  AxisIdle,

  NciControl            := 2000,
  NciStartUp,
  NciCycle,
  NciIdle,
  NciJob,

  FlyingSawControl      := 2100,
  FlyingSawStartUp,


  StationLinkedList     := 3000,
  StationInitList,
  StationAddHead,
  StationAddTail,
  StationGetHead,
  StationRemoveHeadValue,
  StationGearInDistanceToSync,
  StationGearInSyncStart,
  StationGearInSyncMove,
  StationGearInSyncEnd,
  StationCalcInfeedPosition,

  StationControl        := 4000,
  StationState, 

  Xpu_fbEnvironment     := 5000,
  Xpu_fbProcessingUnit,
  Xpu_fbXpuPart,
  Xpu_fbXpuTrack,
  Xpu_fbMc2CaGroup,
  Xpu_fbParameterSet,
  Xpu_fbNctController,

  Xpu_fbPartModules     := 5500,

  Xpu_fbMoverXpu        := 6000,

  Xpu_fbNctBaseUnit     := 6500,

  TransportUnit_General := 7000,
  TransportUnit_Restart := 7010,
  TransportUnit_Start,
  TransportUnit_XpuInit,
  TransportUnit_StationClearOutfeed,

  CamControl            := 8000,
  CamStartUp,
  CamCycle,

  Process_StationCollector    := 11000,
  Process_ProcessCollector    := 11100,
  Process_ProcessCollector_Init,
  Process_ProcessCollector_Cycle,
  Process_ProcessCollector_Control,

  Process_LinkedList_GetHead,
  Process_LinkedList_RemoveHead,
  Process_LinkedList_AddTail,
  Process_LinkedList_CheckData,
  Process_StationQueue_Check,

  Process_LinkedList_Com              := 11200,
  Process_LinkedList_Com_Init,
  Process_LinkedList_Com_Cmd,
  Process_LinkedList_Com_AddHead,
  Process_LinkedList_Com_AddTail,
  Process_LinkedList_Com_DelHead,
  Process_LinkedList_Com_DelTail,
  Process_LinkedList_Com_GetHead,
  Process_LinkedList_Com_GetTail,


  Instance_Command              := 12000,
  Instance_ProcessConductor,
  Instance_BufferInfeed,
  Instance_Infeed,
  Instance_BufferOutfeed,
  Instance_Outfeed,
  Instance_Sender_Buffer,

  Ticket_LinkedList_Ctrl        := 12100,
  Ticket_LinkedList_Com_Init,
  Ticket_LinkedList_Com_Cmd,
  Ticket_LinkedList_Com_AddHead,
  Ticket_LinkedList_Com_AddTail,
  Ticket_LinkedList_Com_DelHead,
  Ticket_LinkedList_Com_DelTail,
  Ticket_LinkedList_Com_GetHead,
  Ticket_LinkedList_Com_GetTail,
  

  Application                 := 13000,
  Application_Check,
  Application_Clear,
  Application_Cmd,
  Application_Disable,
  Application_Enable,
  Application_Finish,
  Application_Init,
  Application_Proceed,
  Application_Work


)DINT;
END_TYPE

// ---- _MSG/types/ST_Message.TcDUT
TYPE ST_Message :
STRUCT
  eType         : e_MessageType;
  eDevice       : e_Device;
  eSubdevice    : e_SubDevice;
  {attribute 'displaymode':='hex'}
  iErrorNumber  : ULINT;
  tTime         : STRING(24);
  sText         : STRING(127);
END_STRUCT
END_TYPE

// ---- _MSG/types/ST_MESSAGE_CTRL.TcDUT
TYPE ST_MESSAGE_CTRL :
STRUCT
  Cmd         : E_MESSAGE_CTRL;
END_STRUCT
END_TYPE

// ---- _MSG/types/ST_MESSAGE_STATE.TcDUT
TYPE ST_MESSAGE_STATE :
STRUCT
  State         : E_MESSAGE_STATE;  // as always... combined value of Cmd equivalent and e_progress
END_STRUCT
END_TYPE

// ---- PLC_MOTION/NCI/GVL_NCI.TcGVL
{attribute 'qualified_only'}
VAR_GLOBAL
  AxisConfig                  : ARRAY[1..MAX_NCI_CH] OF ST_3D_Group;     // NC Axis Id to build NCI group

  ChannelCtrl                 : ARRAY[1..MAX_NCI_CH] OF ST_NCI_CTRL;
  ChannelState                : ARRAY[1..MAX_NCI_CH] OF ST_NCI_STATE;


{IF NOT defined (BSD)}
  {info 'PLC_MOTION_LAYER: WIN'}
  ProgramName                 : ARRAY[1..MAX_NCI_CH] OF STRING(255):= ['C:\TwinCAT\Mc\Nci\Test_GST.nc'];
{ELSE}
  {info 'PLC_MOTION_LAYER: BSD'}
  ProgramName                 : ARRAY[1..MAX_NCI_CH] OF STRING(255):= ['/usr/local/etc/TwinCAT/Mc/Nci/Test_GST.nc'];
{END_IF}

  ProgramNameActive           : ARRAY[1..MAX_NCI_CH] OF STRING(255);

  R_ParameterRead             : ARRAY[1..MAX_NCI_CH] OF ST_R_Parameter;
  R_ParameterWrite            : ARRAY[1..MAX_NCI_CH] OF ST_R_Parameter;

  M_FunctionCyclic            : ARRAY[1..MAX_NCI_CH] OF ST_NCI_M_FUNC; // scope variable for M function tests

{IF defined (NCI)}
  {info 'PLC_MOTION_LAYER: NCI'}
  NciCtrl                     : ARRAY[1..MAX_NCI_CH] OF FB_NciChannelCtrl;
{ELSE}
  NciCtrl                     : ARRAY[1..MAX_NCI_CH] OF I_Nci_Ctrl;
{END_IF}
END_VAR

// ---- PLC_MOTION/_GVL/PLC_CONSTANT.TcGVL
//{attribute 'qualified_only'}
VAR_GLOBAL CONSTANT
  //-----------------------------------------------------------------------------
  //-----------------------------------------------------------------------------
  //-----------------------------------------------------------------------------
  // AXIS related limits
  //-----------------------------------------------------------------------------
  MAX_AXIS              : UINT    := 6;
  MAX_RETRY             : UINT    := 5;


  //-----------------------------------------------------------------------------
  // NCI related limits and *.nc standard folder
  //-----------------------------------------------------------------------------
{IF NOT defined (BSD)}
  NCI_DIR               : STRING  := 'C:\TwinCAT\Mc\Nci\';
{ELSE}
  NCI_DIR               : STRING  := '/usr/local/etc/TwinCAT/Mc/Nci/';
{END_IF}

{IF defined (NCI)}
  {info 'PLC_MOTION_LAYER: NCI'}
  NCI_ACTIVE            : BOOL    := TRUE;
  CONFIG_NAME           : STRING  := 'NCI_Spec_Ch_';
{ELSE}
  NCI_ACTIVE            : BOOL    := FALSE;
  CONFIG_NAME           : STRING  := 'NCI_NOT_ACTIVE';
{END_IF}

  MAX_NCI_CH            : UINT    := 1;

  MAX_PATH_STEPS        : UINT    := 5;
  MAX_MC_AXIS           : UINT    := 3;
  MAX_AUX_AXIS          : UINT    := 2;
  MAX_R_PARA            : UINT    := 10;


  //-----------------------------------------------------------------------------
  // CAMMING related limits
  //-----------------------------------------------------------------------------
{IF defined (CAM)}
  {info 'PLC_MOTION_LAYER: CAM'}
  CAM_ACTIVE                  : BOOL    := TRUE;
{ELSE}
  CAM_ACTIVE                  : BOOL    := FALSE;
{END_IF}

  MAX_CAM_CH                  : UINT    := 1;

  MAX_MOTION_FUNCTION_POINTS  : UINT    := 10;

  // HAUD
  // 17.07.2024
  // Start Implementation of Position Trigger function
  //  - Timestamp/position output
  //  - Latch DC time from input
  
  MAX_TRIGGER_BOX             : UINT := 12;
  MAX_TOUCH_PROBE             : UINT := 12;
  MAX_TRIGGER_COUNT           : UINT :=  4;
  MAX_MTI_CH                  : UINT :=  1; // MAX mti channel per EL terminal

{IF defined (XFC)}
  {info 'PLC_MOTION_LAYER: XFC'}
  XFC_ACTIVE                  : BOOL := TRUE;
{ELSE}
  XFC_ACTIVE                  : BOOL := FALSE;
{END_IF}

  // HAUD
  // 2026 05 28
  // Gear In Pos implementation for flying saw application 

{IF defined (SAW)}
  {info 'PLC_MOTION_LAYER: FLYING_SAW'}
  FLY_SAW_ACTIVE              : BOOL  := TRUE;
{ELSE}
  FLY_SAW_ACTIVE              : BOOL  := FALSE;
{END_IF}
END_VAR

// ---- PLC_MOTION/_GVL/PLC_VERSION.TcGVL
{attribute 'qualified_only'}
VAR_GLOBAL CONSTANT
  VERSION               : STRING := 'V 01.01.02';
  // 2026 08 25
  //  - buffered command reset
  //  - clear for one cycle after Halt
  //  - refactoring of ST_MOVE_DATA to ST_AXIS_MOVE_DATA

  // 2026 07 25
  //  - OS testing concluded
  //  - refactoring update to facilitate easier merge with XTS_TRANSPORT_LAYER into one code base (if you wish to do so)

  // 2026 07 24
  // folder structure changed
  //  - classes , programs and gvl data are now in the same folder
  //
  // messaging unified with XTS_TRANSPORT_LAYER
  //  - f_MessageSet now equal across codebase
  //  - placeholder data for XTS added
  //  - renaming of programs to facilitate merge with XTS_TRANSPORT_LAYER
  //  - UTC time and timezone offset
  //    - timezone timestamp is now used for messaging

  // 2026 05 28 HAUD
  // Flying Saw wrapper

  // 2026 05 13 HAUD
  //
  // FB_McAxisBase.MoveVeloBuffer Test, changes for setpoint change detection

  // 2025 10 24 HAUD
  //
  // documentation added, 
  // project dev changed to 4026.19
  // Ambiguities resoved

  // 2025 08 21 HAUD
  //
  // e_Device: Application added
  // e_Subdevices: merge with XTS_TRANSPORT_LAYER
  // FB_McAxis: testing SendToPos, distance added to method interface

  // 2025 02 17 HAUD
  //
  // code review
  // Message Levels are set during initialization
  // sizeof mapping data is fetched at startup only

  // 2025 01 09 HAUD
  //
  // - FUNCTIONS
  //    - code review
  //    - ctrl/state mechanic harmonized
  // - MAPPING
  //    - UNIONS added

  // 2024 08 08 HAUD
  //
  // - TC_PLC_MOTION_LAYER: 
  //    - XFC base class added
  //    - TriggerBox (DC output set, DC Input latch)
  //    - TouchProbe (DC Input latch: positive, negative)

  // 2024 06 21 HAUD
  //
  // - TC_PLC_MOTION_LAYER: 
  //    - E_PROGRESS refactoring to match TC_XTS_TRANSPORT_LAYER
  

  // 2024 06 10 HAUD
  //
  // - TC_PLC_MOTION_LAYER: 
  //    - rename repository
  //    - remove LEGACY compatibility
  //
  // - PLC_OPEN_DRIVE:
  //    - deprecated


  // 2024 05 31 HAUD
  // 
  // V 01.00.02
  // precompiler defines: 
  //  - BSD: 
  //    - Tc-BSD file system is used else Windows file system is used
  //
  //  - TEST:
  //    - GVL_MSG.MessageLevel
  // Axis, Cam, Nci have individual message levels now

  // 2024 03 09 HAUD
  // 
  // V 01.00.01
  // MC PtP - execution layer with optional mapping
  // NCI    - execution layer with optional mapping
  // CAM    . execution layer with optional mapping
  // precompiler defines: 
  //  - WIN: windows file system is used else Tc-BSD file system is used
  //  - NCI: NCI libraries are linked in project
  //  - CAM: Camming libraries are linked in project
  //  - AXIS_MAP: mapping is used


  // 2024 02 15 HAUD
  // 
  // V 00.50.04
  //
  // Buffered moves test
  // CamIn Test --> TODO MultiCam
  // Message system, cyclic check for write
  

  // 2024 01 12 HAUD
  //
  // V 00.50.03
  //
  // Building is done
  // start of UnitTesting

  // 2024 01 17 HAUD
  //
  // V 00.50.02
  // 
  // start camming implementation (MC_CamIn_V2)
  // legacy namespace available for downward compatibility of ADS Symbol names

  // 2023 12 23 HAUD
  // NC_PTP
  // - redesign for PLC_OPEN_DRIVE started 
  //    --> E_PROGRESS for state feedback
  // - FB_AxisControl inherits FB_McAxis


  //  2023 10 19
  //  HAUD
  // first draft 
  // TODO: everything

END_VAR

// ---- _MSG/GVL_MSG_XTS.TcGVL
{attribute 'qualified_only'}
VAR_GLOBAL CONSTANT
  //-----------------------------------------------------------------------------
  // file paths for message system
  //  - compiler define option WIN switches to Windows file paths
  //-----------------------------------------------------------------------------
{IF NOT defined (BSD)}
  {info 'WIN folders'}
  LOG_DIR               : STRING  := 'C:\TwinCAT\#MsgFiles\';       // delimiter at the end is mandatory!!
  CON_DIR               : STRING  := 'C:\TwinCAT\#Configuration\';  // delimiter at the end is mandatory!!
{ELSE}
  {info 'BSD folders'}
  LOG_DIR               : STRING  := '/usr/local/etc/TwinCAT/#MsgFiles/';       // delimiter at the end is mandatory!!
  CON_DIR               : STRING  := '/usr/local/etc/TwinCAT/#Configuration/';  // delimiter at the end is mandatory!!
{END_IF}

  LOG_FILE              : STRING  := 'MSG_XtsTransport_';
  LOG_FILE_APP          : STRING  := 'MSG_Application_';
  LOG_FILE_METRIC       : STRING  := 'MSG_XtsTransportMetrics_';

  MAX_MESSAGE           : UINT    := 2000; // max entry in message list
END_VAR
VAR_GLOBAL
  //-----------------------------------------------------------------------------
  // Message System
  //  - Everybody uses f_MessageSet(ST_Message)
  //    - DECISION WHICH LIST IS MADE IN f_MessageSet !!
  //    - which list to use is determined by e_Device in your message
  //
  //  - MessageData instances are self sufficient and need only 
  //    datafield assignment for correct data-flow
  //
  //
  //-----------------------------------------------------------------------------
  //-----------------------------------------------------------------------------
  //-----------------------------------------------------------------------------
  // (ST_Message.eDevice := e_Device.Application)
  //----------------------------------------------------------------------------- 
  ApplicationMessageData          : fb_MessageDataCtrl;
  ApplicationMessageCtrl          : st_message_ctrl;
  ApplicationMessageState         : st_message_state;

  ApplicationMessages             : ARRAY[1..MAX_MESSAGE] OF ST_Message;
  MessageApplicationIndex         : UINT := 0; // message index for higher layers (grouping, Instances, etc.)
  MessageApplicationError         : UINT := 0; // error counter for higher learning
  //-----------------------------------------------------------------------------
  //-----------------------------------------------------------------------------
  // (ST_Message.eDevice := from Device_Null to XfcAxis)
  //-----------------------------------------------------------------------------
  TransportMessageData            : fb_MessageDataCtrl;
  TransportMessageCtrl            : st_message_ctrl;
  TransportMessageState           : st_message_state;

  TransportMessages               : ARRAY[1..MAX_MESSAGE] OF ST_Message;
  MessageTransportIndex           : UINT := 0; // message index for base layer
  MessageTransportError           : UINT := 0; // error counter for base layer
  //-----------------------------------------------------------------------------
  //-----------------------------------------------------------------------------
  // (ST_Message.eDevice := e_Device.Metrics)
  //-----------------------------------------------------------------------------
  MetricsMessageData              : fb_MessageDataCtrl;
  MetricsMessageCtrl              : st_message_ctrl;
  MetricsMessageState             : st_message_state;

  MetricsMessages                 : ARRAY[1..MAX_MESSAGE] OF ST_Message;
  MessageMetricsIndex             : UINT := 0; // message index for metrics data
  MessageMetricsError             : UINT := 0; // error counter for metrics data
  //-----------------------------------------------------------------------------
  //-----------------------------------------------------------------------------
  // (ST_Message.eDevice := e_Device.ProductData)
  //-----------------------------------------------------------------------------
  ProductMessageData              : fb_MessageDataCtrl;   // This is for you
  ProductMessageCtrl              : st_message_ctrl;
  ProductMessageState             : st_message_state;

  ProductMessages                 : ARRAY[1..MAX_MESSAGE] OF ST_Message;
  MessageProductIndex             : UINT := 0; // message index for your product data
  MessageProductError             : UINT := 0; // error counter for your product data
  //-----------------------------------------------------------------------------
  //-----------------------------------------------------------------------------
  fbLocalTime                     : fb_LocalTime;
  dtLocalTime                     : DT;
  sLocalTime                      : STRING;
  //-----------------------------------------------------------------------------
  //-----------------------------------------------------------------------------
  //-----------------------------------------------------------------------------
  //-----------------------------------------------------------------------------
  MessageLevelXpu                 : E_MessageType;
  MessageLevelStations            : ARRAY[1..MAX_STATION] OF E_MessageType;
  MessageLevelMovers              : ARRAY[1..MAX_MOVER]   OF E_MessageType;

  MessageLevelProcess             : ARRAY[1..MAX_PROCESS] OF E_MessageType;

{IF defined (TEST)}
  {info 'TEST logging enabled'}
  MessageLevel                    : E_MessageType := eMessageinfo; // a lot of messages
{ELSE}
  MessageLevel                    : E_MessageType := eMessageEmpty; // only errors are written into list 
{END_IF}

END_VAR

// ---- _MSG/GVL_MSG_AXIS.TcGVL
{attribute 'qualified_only'}
VAR_GLOBAL CONSTANT
  //-----------------------------------------------------------------------------
  // file paths for message system
  //  - compiler define option WIN switches to Windows file paths
  //-----------------------------------------------------------------------------
{IF NOT defined (BSD)}
  {info 'PLC_MOTION_LAYER: WIN'}
  LOG_DIR               : STRING  := 'C:\TwinCAT\#MsgFiles\';
{ELSE}
  {info 'PLC_MOTION_LAYER: BSD'}
  LOG_DIR               : STRING  := '/usr/local/etc/TwinCAT/#MsgFiles/';
{END_IF}

  LOG_FILE              : STRING  := concat(TO_STRING(TwinCAT_SystemInfoVarList._AppInfo.AdsPort), '_MSG_PLC_');
  LOG_FILE_METRIC       : STRING  := concat(TO_STRING(TwinCAT_SystemInfoVarList._AppInfo.AdsPort), '_MSG_Metrics_');

  MAX_MESSAGE           : UINT    := 200; // max entry in message list
END_VAR
VAR_GLOBAL
  //-----------------------------------------------------------------------------
  // Message System
  //  - Everybody uses f_MessageSet(ST_Message)
  //    - DECISION WHICH LIST IS MADE IN f_MessageSet !!
  //    - which list to use is determined by e_Device in your message
  //
  //  - MessageData instances are self sufficient and need only 
  //    datafield assignment for correct data-flow
  //
  //
  //-----------------------------------------------------------------------------
  //-----------------------------------------------------------------------------
  //-----------------------------------------------------------------------------
  // (ST_Message.eDevice := from Device_Null to XfcAxis)
  //-----------------------------------------------------------------------------
  MotionMessageData               : fb_MessageDataCtrl;
  MotionMessageCtrl               : st_message_ctrl;
  MotionMessageState              : st_message_state;

  MotionMessages                  : ARRAY[1..MAX_MESSAGE] OF ST_Message;
  MessageMotionIndex              : UINT := 0; // message index for base layer
  MessageMotionError              : UINT := 0; // error counter for base layer
  //-----------------------------------------------------------------------------
  //-----------------------------------------------------------------------------
  // (ST_Message.eDevice := e_Device.Metrics)
  //-----------------------------------------------------------------------------
  MetricMessageData               : fb_MessageDataCtrl;
  MetricMessageCtrl               : st_message_ctrl;
  MetricMessageState              : st_message_state;

  MetricMessages                  : ARRAY[1..MAX_MESSAGE] OF ST_Message;
  MessageMetricIndex              : UINT := 0; // message index for metrics data
  MessageMetricError              : UINT := 0; // error counter for metrics data
  //-----------------------------------------------------------------------------
  //-----------------------------------------------------------------------------
  fbLocalTime                     : fb_LocalTime;
  dtLocalTime                     : DT;
  sLocalTime                      : STRING;
  //-----------------------------------------------------------------------------
  //-----------------------------------------------------------------------------
  //-----------------------------------------------------------------------------
  //-----------------------------------------------------------------------------
{IF defined (TEST)}
  {info 'TEST logging enabled'}
  MessageLevel                    : E_MessageType := eMessageverbose; // a lot of messages
{ELSE}
  MessageLevel                    : E_MessageType := eMessageEmpty; // only errors are written into list 
{END_IF}

  MessageLevelAxisPtp             : ARRAY[1..PLC_CONSTANT.MAX_AXIS]   OF E_MessageType;
  MessageLevelAxisCam             : ARRAY[1..PLC_CONSTANT.MAX_AXIS]   OF E_MessageType;
  MessageLevelAxisFly             : ARRAY[1..PLC_CONSTANT.MAX_AXIS]   OF E_MessageType;
  MessageLevelNciChn              : ARRAY[1..PLC_CONSTANT.MAX_NCI_CH] OF E_MessageType;

  MessageLevelTriggerBox          : ARRAY[1..PLC_CONSTANT.MAX_TRIGGER_BOX]  OF E_MessageType;
  MessageLevelTouchProbe          : ARRAY[1..PLC_CONSTANT.MAX_TOUCH_PROBE]  OF E_MessageType;


  // diag data
  dbg_AxisIdxGearIn               : ARRAY[1..PLC_CONSTANT.MAX_AXIS]      OF BYTE; // diag for Axis gear in
  dbg_AxisIdxGearInMultiMaster    : ARRAY[1..PLC_CONSTANT.MAX_AXIS,1..4] OF BYTE; // diag for Axis gear in multi master
  dbg_AxisIdxCamIn                : ARRAY[1..PLC_CONSTANT.MAX_AXIS]      OF BYTE; // diag for Axis cam in
END_VAR

// ---- APPLICATION/_types/LinkedList/I_Process_LinkedList.TcIO
INTERFACE I_Process_LinkedList

METHOD AddHeadValue : ST_PROCESS_LIST_RESULT
VAR_INPUT
  stData        : ST_PROCESS_DATA;
END_VAR
END_METHOD

METHOD AddTailValue : ST_PROCESS_LIST_RESULT
VAR_INPUT
  stData        : ST_PROCESS_DATA;
END_VAR
END_METHOD

PROPERTY Count : UDINT
GET
END_GET
END_PROPERTY

PROPERTY Data : ARRAY[1..MAX_LIST_NODES] OF ST_PROCESS_DATA
GET
END_GET
END_PROPERTY

PROPERTY Free : UDINT
GET
END_GET
END_PROPERTY

METHOD GetHead : ST_PROCESS_LIST_RESULT
VAR_INPUT
END_VAR
END_METHOD

METHOD GetTail : ST_PROCESS_LIST_RESULT
VAR_INPUT
END_VAR
VAR
END_VAR
END_METHOD

METHOD InitList : BOOL
END_METHOD

PROPERTY Nodes : ARRAY[0..MAX_LIST_NODES] OF T_LinkedListEntry
GET
END_GET
END_PROPERTY

METHOD RemoveHeadValue : ST_PROCESS_LIST_RESULT
VAR_INPUT
END_VAR
END_METHOD

METHOD RemoveTailValue : ST_PROCESS_LIST_RESULT
VAR_INPUT
END_VAR
VAR
END_VAR
END_METHOD

END_INTERFACE

// ---- PLC_MOTION/FLYING_SAW/class/I_Fly_Ctrl.TcIO
INTERFACE I_Fly_Ctrl

PROPERTY AxisCtrl : pointer to ARRAY[1..PLC_CONSTANT.MAX_AXIS] OF ST_FLY_CTRL
SET
END_SET
END_PROPERTY

PROPERTY AxisIndex : uint
SET
END_SET
END_PROPERTY

PROPERTY AxisModulo : lreal
SET
END_SET
END_PROPERTY

PROPERTY AxisState : pointer to ARRAY[1..PLC_CONSTANT.MAX_AXIS] OF ST_FLY_STATE
SET
END_SET
END_PROPERTY

METHOD Cycle  : e_progress
END_METHOD

PROPERTY GearData : pointer to ARRAY[1..PLC_CONSTANT.MAX_AXIS] OF ST_FLY_DATA
SET
END_SET
END_PROPERTY

PROPERTY ItfMcAxes : array[1..MAX_AXIS] of I_McAxis
SET
END_SET
END_PROPERTY

PROPERTY MessageLevel : E_MessageType
SET
END_SET
END_PROPERTY

PROPERTY MoveData : pointer to ARRAY[1..PLC_CONSTANT.MAX_AXIS] OF ST_AXIS_MOVE_DATA
SET
END_SET
END_PROPERTY

PROPERTY Options : pointer to ARRAY[1..PLC_CONSTANT.MAX_AXIS] OF ST_FLY_OPTIONS
SET
END_SET
END_PROPERTY

END_INTERFACE

// ---- PLC_MOTION/NCI/class/I_Nci_Ctrl.TcIO
INTERFACE I_Nci_Ctrl

PROPERTY ChnCtrl : pointer to ST_NCI_CTRL
SET
END_SET
END_PROPERTY

PROPERTY ChnId : udint
GET
END_GET
END_PROPERTY

PROPERTY ChnState : pointer to ST_NCI_STATE
SET
END_SET
END_PROPERTY

METHOD Cycle : E_PROGRESS
VAR_INPUT
END_VAR
END_METHOD

PROPERTY ItfChannel : I_NciChannel
GET
END_GET
END_PROPERTY

PROPERTY M_FunctionScope : pointer to st_nci_m_func
SET
END_SET
END_PROPERTY

END_INTERFACE

// ---- _MSG/I_MessageData.TcIO
INTERFACE I_MessageData

PROPERTY DirRoot : POINTER to string(255)
SET
END_SET
END_PROPERTY

PROPERTY ErrorIndex : reference to uint
SET
END_SET
END_PROPERTY

PROPERTY FileRoot : pointer to string(255)
SET
END_SET
END_PROPERTY

PROPERTY LocalTime : pointer to DT
SET
END_SET
END_PROPERTY

PROPERTY MessageIndex : reference to uint
SET
END_SET
END_PROPERTY

PROPERTY MsgList : pointer to ARRAY[1..GVL_MSG_AXIS.MAX_MESSAGE] OF st_message
SET
END_SET
END_PROPERTY

END_INTERFACE

// ---- MAPPING/MAPPING_AXIS_in.TcPOU
PROGRAM MAPPING_AXIS_in
VAR CONSTANT
//-----------------------------------------------------------------------------------------------------------------
//  Stop! Who approacheth the Bridge of Death must answer me these questions three, ere the other side he see
//-----------------------------------------------------------------------------------------------------------------
{IF defined (AXIS_MAP)}
  {info 'PLC_MOTION_LAYER: AXIS_MAP'}
  bBypassMappingAxis        : BOOL  := FALSE;
{ELSE}
  bBypassMappingAxis        : BOOL  := TRUE;
{END_IF}
//-----------------------------------------------------------------------------------------------------------------
//  What... is your name?
//-----------------------------------------------------------------------------------------------------------------
{IF defined (NCI_MAP)}
  {info 'PLC_MOTION_LAYER: NCI_MAP'}
  bBypassMappingNci         : BOOL  := FALSE;
{ELSE}
  bBypassMappingNci         : BOOL  := TRUE;
{END_IF}
//-----------------------------------------------------------------------------------------------------------------
//  What... is your quest?
//-----------------------------------------------------------------------------------------------------------------
{IF defined (CAM_MAP)}
  {info 'PLC_MOTION_LAYER: CAM_MAP'}
  bBypassMappingCam         : BOOL  := FALSE;
{ELSE}
  bBypassMappingCam         : BOOL  := TRUE;
{END_IF}
{IF defined (SAW_MAP)}
  {info 'PLC_MOTION_LAYER: SAW_MAP'}
  bBypassMappingFlyingSaw   : BOOL  := FALSE;
{ELSE}
  bBypassMappingFlyingSaw   : BOOL  := TRUE;
{END_IF}
//-----------------------------------------------------------------------------------------------------------------
//  What... is the capital of Assyria?
//-----------------------------------------------------------------------------------------------------------------
{IF defined (TRIGGER_MAP)}
  {info 'PLC_MOTION_LAYER: TRIGGER_MAP'}
  bBypassMappingTrigger     : BOOL  := FALSE;
{ELSE}
  bBypassMappingTrigger     : BOOL  := TRUE;
{END_IF}
END_VAR
VAR
  sMappingCheck             : STRING;
//-----------------------------------------------------------------------------------------------------------------
//  Ask me the questions, bridgekeeper. I'm not afraid.
//-----------------------------------------------------------------------------------------------------------------
{IF defined (AXIS_MAP)}
  AxisCtrl                  : U_AXIS_CTRL;
  AxisMoveData              : U_AXIS_MOVE_DATA;
  AxisMotionOptions         : U_AXIS_MOTION_OPTIONS;

  AxisGearInData            : U_AXIS_GEAR_IN;
  AxisHoming                : U_AXIS_HOMING;
  AxisParameterIn           : U_AXIS_NC_PARAMETER_WRT;

  SelectorCtrl              : U_PARAMETER_SELECTOR_CTRL;
{ELSE}
  AxisCtrl                  : BYTE;
  AxisMoveData              : BYTE;
  AxisMotionOptions         : BYTE;

  AxisGearInData            : BYTE;
  AxisHoming                : BYTE;
  AxisParameterIn           : BYTE;

  SelectorCtrl              : byte;
{END_IF}
//-----------------------------------------------------------------------------------------------------------------
//  Sir Robin of Camelot.
//-----------------------------------------------------------------------------------------------------------------
{IF defined (NCI_MAP)}
  NciControl                : U_NCI_CTRL;
  NciAxisGroup              : U_NCI_AXIS_ID_GROUP;
  NciRparameters            : U_NCI_R_PARAMETER_I;
{ELSE}
  NciControl                : BYTE;
  NciAxisGroup              : BYTE;
  NciRparameters            : BYTE;
{END_IF}
//-----------------------------------------------------------------------------------------------------------------
//  To seek the Holy Grail.
//-----------------------------------------------------------------------------------------------------------------
{IF defined (CAM_MAP)}
  CamControl                : U_CAM_CTRL;
  CamData                   : U_CAM_DATA;
{ELSE}
  CamControl                : BYTE;
  CamData                   : byte;
{END_IF}
//-----------------------------------------------------------------------------------------------------------------
//  .....
//-----------------------------------------------------------------------------------------------------------------
{IF defined (TRIGGER_MAP)}
  TriggerControl            : U_TRIGGER_CTRL;
  TouchProbeControl         : U_TOUCH_PROBE_CTRL;
{ELSE}
  //  I don't know that! Auuuuuuuugh!
  TriggerControl            : BYTE;
  TouchProbeControl         : BYTE;
{END_IF}
//-----------------------------------------------------------------------------------------------------------------
//  .....
//-----------------------------------------------------------------------------------------------------------------
{IF defined (SAW_MAP)}
  FlyControl                : U_FLY_CTRL;
  FlyData                   : U_FLY_DATA;
  FlyOptions                : U_FLY_OPTIONS;
{ELSE}
  //  I don't know that! Auuuuuuuugh!
  FlyControl                : byte;
  FlyData                   : byte;
  FlyOptions                : BYTE;
{END_IF}
//-----------------------------------------------------------------------------------------------------------------
//   What... is the air-speed velocity of an unladen swallow?
//-----------------------------------------------------------------------------------------------------------------
  bMappingBlocked           : BOOL;   //  How do know so much about swallows?
//-----------------------------------------------------------------------------------------------------------------
//  - datafield size check
//-----------------------------------------------------------------------------------------------------------------
  szSelectorCtrl,
  szAxisPara,
  szAxisHoming,
  szAxisGearData,
  szAxisMotionOptions,
  szAxisMoveData,
  szAxisCtrl                : ARRAY[1..2] OF UDINT;

  szNciRparameters,
  szNciAxisGroup,
  szNciCtrl                 : ARRAY[1..2] OF UDINT;

  szCamCtrl                 : ARRAY[1..2] OF UDINT;

  szCtrlTouchProbe,
  szCtrlTrigger             : ARRAY[1..2] OF UDINT;

  szFlyingSawCtrl,
  szFlyingSawData,
  szFlyingSawOptions        : ARRAY[1..2] OF UDINT;
END_VAR

//-----------------------------------------------------------------------------------------------------------------
//  - datafield size check
//-----------------------------------------------------------------------------------------------------------------
IF NOT Check() THEN RETURN; END_IF
//--------------------------------------------------------------------------------------------
//--------------------------------------------------------------------------------------------
//  What do you mean? An African or European swallow?
//--------------------------------------------------------------------------------------------
IF bMappingBlocked
THEN
  RETURN; // Huh? I-- I don't know that. Auuuuuuuugh!
END_IF
//--------------------------------------------------------------------------------------------
//  Well, you have to know these things when you're a king, you know.
//--------------------------------------------------------------------------------------------
//--------------------------------------------------------------------------------------------
//           destination,                         source,                      size
//--------------------------------------------------------------------------------------------
IF NOT bBypassMappingAxis
THEN
  memcpy(ADR(GVL_AXIS.Ctrl),                 ADR(AxisCtrl),             SIZEOF(AxisCTrl));
  memcpy(ADR(GVL_AXIS.Data),                 ADR(AxisMoveData),         SIZEOF(AxisMoveData));
  memcpy(ADR(GVL_AXIS.MotionOptions),        ADR(AxisMotionOptions),    SIZEOF(AxisMotionOptions));

  memcpy(ADR(GVL_AXIS.GearInParameter),      ADR(AxisGearInData),       SIZEOF(AxisGearInData));
  memcpy(ADR(GVL_AXIS.HomeParameter),        ADR(AxisHoming),           SIZEOF(AxisHoming));
  memcpy(ADR(GVL_AXIS.NcParameterIn),        ADR(AxisParameterIn),      SIZEOF(AxisParameterIn));

  memcpy(ADR(GVL_AXIS.SelectorCtrl),         ADR(SelectorCtrl),         SIZEOF(SelectorCtrl));
END_IF
//--------------------------------------------------------------------------------------------
//--------------------------------------------------------------------------------------------
IF NOT bBypassMappingNci
THEN
  memcpy(ADR(GVL_NCI.ChannelCtrl),           ADR(NciControl),           SIZEOF(NciControl));
  memcpy(ADR(GVL_NCI.AxisConfig),            ADR(NciAxisGroup),         SIZEOF(NciAxisGroup));
  memcpy(ADR(GVL_NCI.R_ParameterWrite),      ADR(NciRparameters),       SIZEOF(NciRparameters));
END_IF
//--------------------------------------------------------------------------------------------
//--------------------------------------------------------------------------------------------
IF NOT bBypassMappingCam
THEN
  memcpy(ADR(GVL_CAM.Ctrl),                  ADR(CamControl),           SIZEOF(CamControl));
  memcpy(ADR(GVL_CAM.Data),                  ADR(CamData),              SIZEOF(CamData));
END_IF
//--------------------------------------------------------------------------------------------
//--------------------------------------------------------------------------------------------
IF NOT bBypassMappingTrigger
THEN
  memcpy(ADR(GVL_FUNCTIONS.CtrlTrigger),     ADR(TriggerControl),       SIZEOF(TriggerControl));
  memcpy(ADR(GVL_FUNCTIONS.CtrlTouchProbe),  ADR(TouchProbeControl),    SIZEOF(TouchProbeControl));
END_IF
//--------------------------------------------------------------------------------------------
//--------------------------------------------------------------------------------------------
IF NOT bBypassMappingFlyingSaw
THEN
  memcpy(ADR(GVL_FLYING_SAW.Ctrl),          ADR(FlyControl),            SIZEOF(FlyControl));
  memcpy(ADR(GVL_FLYING_SAW.Data),          ADR(FlyData),               SIZEOF(FlyData));
  memcpy(ADR(GVL_FLYING_SAW.Options),       ADR(FlyOptions),            SIZEOF(FlyOptions));
END_IF
//--------------------------------------------------------------------------------------------
//--------------------------------------------------------------------------------------------
//           destination,                         source,                      size
//--------------------------------------------------------------------------------------------

METHOD Check : bool
//--------------------------------------------------------------------------------------------
//--------------------------------------------------------------------------------------------
IF bBypassMappingAxis AND
   bBypassMappingNci  AND
   bBypassMappingCam  AND
   bBypassMappingTrigger AND
   bBypassMappingFlyingSaw
THEN
  sMappingCheck         := 'NO_MAPPING_ACTIVE';
  RETURN;
END_IF
//--------------------------------------------------------------------------------------------
//--------------------------------------------------------------------------------------------
szAxisCtrl[1]           := SIZEOF(AxisCtrl);
szAxisCtrl[2]           := SIZEOF(GVL_AXIS.Ctrl);

szAxisMoveData [1]      := SIZEOF(AxisMoveData);
szAxisMoveData [2]      := SIZEOF(GVL_AXIS.Data);

szAxisMotionOptions [1] := SIZEOF(AxisMotionOptions);
szAxisMotionOptions [2] := SIZEOF(GVL_AXIS.MotionOptions);

szAxisGearData [1]      := SIZEOF(AxisGearInData);
szAxisGearData [2]      := SIZEOF(GVL_AXIS.GearInParameter);

szAxisHoming [1]        := SIZEOF(AxisHoming);
szAxisHoming [2]        := SIZEOF(GVL_AXIS.HomeParameter);

szAxisPara [1]          := SIZEOF(AxisParameterIn);
szAxisPara [2]          := SIZEOF(GVL_AXIS.NcParameterIn);

szSelectorCtrl[1]       := SIZEOF(SelectorCtrl);
szSelectorCtrl[2]       := SIZEOF(GVL_AXIS.SelectorCtrl);

IF NOT (bBypassMappingAxis)
THEN
  IF NOT (szAxisCtrl[1] = szAxisCtrl[2])
  THEN
    sMappingCheck       := 'AxisCtrl CHECK_ERROR';
    RETURN;
  END_IF

  IF NOT (szAxisMoveData[1] = szAxisMoveData[2])
  THEN
    sMappingCheck       := 'AxisMoveData CHECK_ERROR';
    RETURN;
  END_IF

  IF NOT (szAxisMotionOptions[1] = szAxisMotionOptions[2])
  THEN
    sMappingCheck       := 'AxisMotionOptions CHECK_ERROR';
    RETURN;
  END_IF

  IF NOT (szAxisGearData[1] = szAxisGearData[2])
  THEN
    sMappingCheck       := 'AxisGearInData CHECK_ERROR';
    RETURN;
  END_IF

  IF NOT (szAxisHoming[1] = szAxisHoming[2])
  THEN
    sMappingCheck       := 'AxisHoming CHECK_ERROR';
    RETURN;
  END_IF

  IF NOT (szSelectorCtrl[1] = szSelectorCtrl[2])
  THEN
    sMappingCheck       := 'SelectorCtrl CHECK_ERROR';
    return;
  END_IF
END_IF
//--------------------------------------------------------------------------------------------
//--------------------------------------------------------------------------------------------
szNciCtrl[1]            := SIZEOF(NciControl);
szNciCtrl[2]            := SIZEOF(GVL_NCI.ChannelCtrl);

szNciAxisGroup  [1]     := SIZEOF(NciAxisGroup);
szNciAxisGroup  [2]     := SIZEOF(GVL_NCI.AxisConfig);

szNciRparameters[1]     := SIZEOF(NciRparameters);
szNciRparameters[2]     := SIZEOF(GVL_NCI.R_ParameterWrite);

IF NOT (bBypassMappingNci)
THEN
  IF NOT (szNciCtrl[1] = szNciCtrl[2])
  THEN
    sMappingCheck       := 'NciControl CHECK_ERROR';
    RETURN;
  END_IF

  IF NOT (szNciAxisGroup[1] = szNciAxisGroup[2])
  THEN
    sMappingCheck       := 'NciAxisGroup CHECK_ERROR';
    RETURN;
  END_IF

  IF NOT (szNciRparameters[1] = szNciRparameters[2])
  THEN
    sMappingCheck       := 'NciRparameters CHECK_ERROR';
    RETURN;
  END_IF
END_IF
//--------------------------------------------------------------------------------------------
//--------------------------------------------------------------------------------------------
szCamCtrl [1]           := SIZEOF(CamControl);
szCamCtrl [2]           := SIZEOF(GVL_CAM.Ctrl);

IF NOT (bBypassMappingCam)
THEN
  IF NOT (szCamCtrl[1] = szCamCtrl[2])
  THEN
    sMappingCheck       := 'CamControl CHECK_ERROR';
    RETURN;
  END_IF
END_IF
//--------------------------------------------------------------------------------------------
//--------------------------------------------------------------------------------------------
szCtrlTrigger[1]        := SIZEOF(TriggerControl);
szCtrlTrigger[2]        := SIZEOF(GVL_FUNCTIONS.CtrlTrigger);

szCtrlTouchProbe[1]     := SIZEOF(TouchProbeControl);
szCtrlTouchProbe[2]     := SIZEOF(GVL_FUNCTIONS.CtrlTouchProbe);

IF NOT (bBypassMappingTrigger)
THEN
  IF NOT (szCtrlTrigger[1] = szCtrlTrigger[2])
  THEN
    sMappingCheck       := 'TriggerControl CHECK_ERROR';
    RETURN;
  END_IF

  IF NOT (szCtrlTouchProbe[1] = szCtrlTouchProbe[2])
  THEN
    sMappingCheck       := 'TouchProbeControl CHECK_ERROR';
    RETURN;
  END_IF
END_IF
//--------------------------------------------------------------------------------------------
//--------------------------------------------------------------------------------------------
szFlyingSawCtrl[1]      := SIZEOF(FlyControl);
szFlyingSawCtrl[2]      := SIZEOF(GVL_FLYING_SAW.Ctrl);

szFlyingSawData[1]      := SIZEOF(FlyData);
szFlyingSawData[2]      := SIZEOF(GVL_FLYING_SAW.Data);

szFlyingSawOptions[1]   := SIZEOF(FlyOptions);
szFlyingSawOptions[2]   := SIZEOF(GVL_FLYING_SAW.Options);

IF NOT (bBypassMappingFlyingSaw)
THEN
  IF NOT (szFlyingSawCtrl[1] = szFlyingSawCtrl[2])
  THEN
    sMappingCheck       := 'FlyControl CHECK_ERROR';
    RETURN;
  END_IF

  IF NOT (szFlyingSawData[1] = szFlyingSawData[2])
  THEN
    sMappingCheck       := 'FlyData CHECK_ERROR';
    RETURN;
  END_IF

  IF NOT (szFlyingSawOptions[1] = szFlyingSawOptions[2])
  THEN
    sMappingCheck       := 'FlyOptions CHECK_ERROR';
    RETURN;
  END_IF
END_IF
//--------------------------------------------------------------------------------------------
//--------------------------------------------------------------------------------------------
//--------------------------------------------------------------------------------------------
//--------------------------------------------------------------------------------------------
sMappingCheck           := 'CHECK_DONE';
Check                   := TRUE;
//--------------------------------------------------------------------------------------------
//--------------------------------------------------------------------------------------------
END_METHOD

END_PROGRAM

// ---- PLC_MOTION/NC_PTP/MAIN_AXIS.TcPOU
PROGRAM MAIN_AXIS
VAR
  eInit         AT %Q*      : E_PROGRESS;   // shall be checked by controlling entity, before using Ctrl/State structs

  nAxis,
  nAxisInit                 : UINT;

  stMsg                   : ST_Message;
  eMsgState               : e_message_state;
  eMsgProgress            : E_PROGRESS;
  eMtrState               : e_message_state;
  eMtrProgress            : E_PROGRESS;

  tIdleWriteMotion        : TIME := T#5S;
  tIdleWriteMetric        : TIME := T#5S;
  tonIdleWriteMotion      : Tc2_Standard.TON;
  tonIdleWriteMetric      : Tc2_Standard.TON;
END_VAR

//-----------------------------------------------------------------------------------------------------------------
// Local time; used for timestamps
//-----------------------------------------------------------------------------------------------------------------
GVL_MSG_AXIS.fbLocalTime();
GVL_MSG_XTS.sLocalTime                            :=
GVL_MSG_AXIS.sLocalTime                       := GVL_MSG_AXIS.fbLocalTime.LocalTimeString;
GVL_MSG_XTS.dtLocalTime                           :=
GVL_MSG_AXIS.dtLocalTime                      := GVL_MSG_AXIS.fbLocalTime.LocalTime;
//-----------------------------------------------------------------------------------------------------------------
// /assign dataflow
//-----------------------------------------------------------------------------------------------------------------
FOR nAxis := 1 TO PLC_CONSTANT.MAX_AXIS
DO
  GVL_AXIS.Control[nAxis].AxisIndex           := nAxis;
  GVL_AXIS.Control[nAxis].MessageLevel        := GVL_MSG_AXIS.MessageLevelAxisPtp[nAxis];

  GVL_AXIS.Control[nAxis].AxisCtrl            := ADR(GVL_AXIS.Ctrl);          // command
  GVL_AXIS.Control[nAxis].AxisState           := ADR(GVL_AXIS.State);         // state + result of command

  GVL_AXIS.Control[nAxis].Axes                REF=   GVL_AXIS.AxisRef;        // All for one; coupling requires access across all axes

  GVL_AXIS.Control[nAxis].AxisInfo            := ADR(GVL_AXIS.Info);          // axis information: act/set values and bits from axis
  GVL_AXIS.Control[nAxis].AxisData            := ADR(GVL_AXIS.Data);          // position and dynamic constraints for movement
  GVL_AXIS.Control[nAxis].AxisGearInParameter := ADR(GVL_AXIS.GearInParameter);

  GVL_AXIS.Control[nAxis].NcParameterOut      := ADR(GVL_AXIS.NcParameterOut);
  GVL_AXIS.Control[nAxis].NcParameterIn       := ADR(GVL_AXIS.NcParameterIn);

  GVL_AXIS.Control[nAxis].HomingParameter     := ADR(GVL_AXIS.HomeParameter);
  GVL_AXIS.Control[nAxis].MotionOptions       := ADR(GVL_AXIS.MotionOptions);
  GVL_AXIS.Control[nAxis].LimitSwitches       := ADR(GVL_AXIS.LimitSwitches);

  GVL_AXIS.ItfMcAxis[nAxis]                   := GVL_AXIS.Control[nAxis]; 
END_FOR

GVL_AXIS.ParameterSelector.MessageLevel       :=   GVL_MSG_XTS.MessageLevel;
GVL_AXIS.ParameterSelector.Ctrl               REF= GVL_AXIS.SelectorCtrl;
GVL_AXIS.ParameterSelector.State              REF= GVL_AXIS.SelectorState;
GVL_AXIS.ParameterSelector.ItfAxis            REF= GVL_AXIS.ItfMcAxis;
//-----------------------------------------------------------------------------------------------------------------
// assign dataflow/
//-----------------------------------------------------------------------------------------------------------------
//-----------------------------------------------------------------------------------------------------------------
//-----------------------------------------------------------------------------------------------------------------
// /INIT
// - successful init is required for other optional members to start
//-----------------------------------------------------------------------------------------------------------------
CASE eInit
OF
  E_PROGRESS.PROGRESS_INVALID:
    GVL_MSG_AXIS.MotionMessageCtrl.Cmd        := E_MESSAGE_CTRL.MSG_CTRL_NULL;
    GVL_MSG_AXIS.MetricMessageCtrl.Cmd        := E_MESSAGE_CTRL.MSG_CTRL_NULL;

    FOR nAxis := 1 TO PLC_CONSTANT.MAX_AXIS
    DO
      GVL_MSG_AXIS.MessageLevelAxisPtp[nAxis] := E_MessageType.eMessageVerbose; //GVL_MSG.MessageLevel;
    END_FOR
    nAxisInit                                 := 1;
    eInit                                     := E_PROGRESS.PROGRESS_INIT;
  //-----------------------------------------------------------------------------
  //-----------------------------------------------------------------------------
  E_PROGRESS.PROGRESS_INIT:
    stMsg.eType                               := E_MessageType.eMessageInfo;
    stMsg.eDevice                             := e_Device.Device_MainAxis;
    stMsg.eSubdevice                          := e_SubDevice.MainInit;
    stMsg.iErrorNumber                        := MAX_AXIS;
    stMsg.sText                               := concat('MAIN_AXIS.eInit: ', TO_STRING(eInit));
    f_MessageSet(stMsg);

    GVL_MSG_AXIS.MotionMessageCtrl.Cmd        := E_MESSAGE_CTRL.MSG_CTRL_INIT;
    GVL_MSG_AXIS.MetricMessageCtrl.Cmd        := E_MESSAGE_CTRL.MSG_CTRL_INIT;
    eInit                                     := E_PROGRESS.PROGRESS_BUSY;
  //-----------------------------------------------------------------------------
  //-----------------------------------------------------------------------------
  E_PROGRESS.PROGRESS_BUSY:
    eInit                                     := E_PROGRESS.PROGRESS_PREPARE;
  //-----------------------------------------------------------------------------
  //-----------------------------------------------------------------------------
  E_PROGRESS.PROGRESS_PREPARE:
    stMsg.eType                               := E_MessageType.eMessageVerbose;
    stMsg.eDevice                             := e_Device.Device_MainAxis;
    stMsg.eSubdevice                          := e_SubDevice.MainInit;
    stMsg.iErrorNumber                        := nAxisInit;
    stMsg.sText                               := concat('AxisInit Index: ', TO_STRING(nAxisInit));

    IF (GVL_MSG_AXIS.MessageLevelAxisPtp[nAxisInit] = E_MessageType.eMessageVerbose)
    THEN
      f_MessageSet(stMsg);
    END_IF

    GVL_AXIS.Ctrl[nAxisInit].eCmd             := E_AXIS_CTRL.AXIS_NULL;
    eInit                                     := E_PROGRESS.PROGRESS_STARTUP;
  //-----------------------------------------------------------------------------
  //-----------------------------------------------------------------------------
  E_PROGRESS.PROGRESS_STARTUP:
    GVL_AXIS.Ctrl[nAxisInit].eCmd             := E_AXIS_CTRL.AXIS_INIT;

    IF    (GVL_AXIS.State[nAxisInit].eState = E_AXIS_STATE.AXIS_INIT + E_PROGRESS.PROGRESS_ERROR)
    THEN
      eInit                                   := E_PROGRESS.PROGRESS_ERROR;

      stMsg.eType                             := E_MessageType.eMessageError;
      stMsg.eDevice                           := e_Device.Device_MainAxis;
      stMsg.eSubdevice                        := e_SubDevice.MainInit;
      stMsg.iErrorNumber                      := GVL_AXIS.Control[nAxisInit].ErrorId;

      stMsg.sText                             := concat('MAIN_AXIS.eInit ERROR at Index: ', TO_STRING(nAxisInit));
      f_MessageSet(stMsg);

    ELSIF (GVL_AXIS.State[nAxisInit].eState = E_AXIS_STATE.AXIS_INIT + E_PROGRESS.PROGRESS_DONE)
    THEN
      eInit                                   := E_PROGRESS.PROGRESS_CHECK;
    END_IF
  //-----------------------------------------------------------------------------
  //-----------------------------------------------------------------------------
  E_PROGRESS.PROGRESS_CHECK:
    IF NOT (nAxisInit > PLC_CONSTANT.MAX_AXIS-1)
    THEN
      nAxisInit                               := nAxisInit + 1;
      eInit                                   := E_PROGRESS.PROGRESS_PREPARE;

    ELSE
      eInit                                   := E_PROGRESS.PROGRESS_OCCUPIED;

      stMsg.eType                             := E_MessageType.eMessageInfo;
      stMsg.eDevice                           := e_Device.Device_MainAxis;
      stMsg.eSubdevice                        := e_SubDevice.MainInit;
      stMsg.iErrorNumber                      := MAX_AXIS;

      stMsg.sText                             := concat('MAIN_AXIS.eInit: ', TO_STRING(E_PROGRESS.PROGRESS_DONE));
      f_MessageSet(stMsg);

      FOR nAxis := 1 TO PLC_CONSTANT.MAX_AXIS
      DO
        GVL_MSG_AXIS.MessageLevelAxisPtp[nAxis]  := GVL_MSG_XTS.MessageLevel;
      END_FOR
    END_IF

  E_PROGRESS.PROGRESS_OCCUPIED:
   eInit                                     := E_PROGRESS.PROGRESS_DONE;
END_CASE
//-----------------------------------------------------------------------------------------------------------------
// INIT/
//-----------------------------------------------------------------------------------------------------------------
//-----------------------------------------------------------------------------------------------------------------
//-----------------------------------------------------------------------------------------------------------------
// /cyclic
//-----------------------------------------------------------------------------------------------------------------
IF (eInit <> E_PROGRESS.PROGRESS_ERROR)
THEN
  FOR nAxis := 1 TO PLC_CONSTANT.MAX_AXIS
  DO
      GVL_AXIS.Control[nAxis]();
  END_FOR

  GVL_AXIS.ParameterSelector();
END_IF
//-----------------------------------------------------------------------------------------------------------------
// cyclic/
//-----------------------------------------------------------------------------------------------------------------
//-----------------------------------------------------------------------------------------------------------------
//  /logging
//    - all life is problem solving
//-----------------------------------------------------------------------------------------------------------------
GVL_MSG_AXIS.MotionMessageData.Ctrl           REF= GVL_MSG_AXIS.MotionMessageCtrl;
GVL_MSG_AXIS.MotionMessageData.State          REF= GVL_MSG_AXIS.MotionMessageState;
GVL_MSG_AXIS.MotionMessageData.MessageIndex   REF= GVL_MSG_AXIS.MessageMotionIndex;
GVL_MSG_AXIS.MotionMessageData.ErrorIndex     REF= GVL_MSG_AXIS.MessageMotionError;
GVL_MSG_AXIS.MotionMessageData.DirRoot        :=   ADR(GVL_MSG_AXIS.LOG_DIR);
GVL_MSG_AXIS.MotionMessageData.FileRoot       :=   ADR(GVL_MSG_AXIS.LOG_FILE);
GVL_MSG_AXIS.MotionMessageData.MsgList        :=   ADR(GVL_MSG_AXIS.MotionMessages);
GVL_MSG_AXIS.MotionMessageData.LocalTime      :=   ADR(GVL_MSG_AXIS.dtLocalTime);
GVL_MSG_AXIS.MotionMessageData();               

eMsgState                                     :=   f_GetState   (GVL_MSG_AXIS.MotionMessageState.State);
eMsgProgress                                  :=   f_GetProgress(GVL_MSG_AXIS.MotionMessageState.State);

CASE eMsgState
OF
  E_MESSAGE_STATE.MSG_STATE_NULL:
    CASE eMsgProgress
    OF
      E_PROGRESS.PROGRESS_INVALID,
      E_PROGRESS.PROGRESS_DONE:
        IF (GVL_MSG_AXIS.MessageMotionIndex > GVL_MSG_XTS.MAX_MESSAGE/100) OR
           (GVL_MSG_AXIS.MessageMotionError > 0)
        THEN
          GVL_MSG_AXIS.MotionMessageCtrl.Cmd  := E_MESSAGE_CTRL.MSG_CTRL_WRITE;
        ELSE
          tonIdleWriteMotion(IN := TRUE, PT:= tIdleWriteMotion);
          IF (tonIdleWriteMotion.Q)
          THEN
            GVL_MSG_AXIS.MotionMessageCtrl.Cmd:= E_MESSAGE_CTRL.MSG_CTRL_WRITE;
          END_IF
        END_IF
    END_CASE

  E_MESSAGE_STATE.MSG_STATE_WRITE:
    CASE eMsgProgress
    OF
      E_PROGRESS.PROGRESS_ERROR,
      E_PROGRESS.PROGRESS_DONE:
        tonIdleWriteMotion(IN := FALSE, PT:= tIdleWriteMotion);
        GVL_MSG_AXIS.MotionMessageCtrl.Cmd    := E_MESSAGE_CTRL.MSG_CTRL_NULL;
    END_CASE

ELSE
    CASE eMsgProgress
    OF
      E_PROGRESS.PROGRESS_DONE:
        GVL_MSG_AXIS.MotionMessageCtrl.Cmd    := E_MESSAGE_CTRL.MSG_CTRL_NULL;
    END_CASE
END_CASE
//-----------------------------------------------------------------------------------------------------------------
//  logging/
//-----------------------------------------------------------------------------------------------------------------
//-----------------------------------------------------------------------------------------------------------------
//-----------------------------------------------------------------------------------------------------------------
//  /Metrics
//-----------------------------------------------------------------------------------------------------------------
GVL_MSG_AXIS.MetricMessageData.Ctrl           REF= GVL_MSG_AXIS.MetricMessageCtrl;
GVL_MSG_AXIS.MetricMessageData.State          REF= GVL_MSG_AXIS.MetricMessageState;

GVL_MSG_AXIS.MetricMessageData.MessageIndex   REF= GVL_MSG_AXIS.MessageMetricIndex;
GVL_MSG_AXIS.MetricMessageData.ErrorIndex     REF= GVL_MSG_AXIS.MessageMetricError;

GVL_MSG_AXIS.MetricMessageData.DirRoot        :=   ADR(GVL_MSG_AXIS.LOG_DIR);
GVL_MSG_AXIS.MetricMessageData.FileRoot       :=   ADR(GVL_MSG_AXIS.LOG_FILE_METRIC);

GVL_MSG_AXIS.MetricMessageData.MsgList        :=   ADR(GVL_MSG_AXIS.MetricMessages);
GVL_MSG_AXIS.MetricMessageData.LocalTime      :=   ADR(GVL_MSG_AXIS.dtLocalTime);

GVL_MSG_AXIS.MetricMessageData();

eMtrState                                     := f_GetState   (GVL_MSG_AXIS.MetricMessageState.State);
eMtrProgress                                  := f_GetProgress(GVL_MSG_AXIS.MetricMessageState.State);

CASE eMtrState
OF
  E_MESSAGE_STATE.MSG_STATE_NULL:
    CASE eMtrProgress
    OF
      E_PROGRESS.PROGRESS_INVALID:
        IF (GVL_MSG_AXIS.MessageMetricIndex > GVL_MSG_XTS.MAX_MESSAGE/100) OR
           (GVL_MSG_AXIS.MessageMetricError > 0)
        THEN
          GVL_MSG_AXIS.MetricMessageCtrl.Cmd  := E_MESSAGE_CTRL.MSG_CTRL_WRITE;
        ELSE
          tonIdleWriteMetric(IN := TRUE, PT:= tIdleWriteMetric);
          IF (tonIdleWriteMetric.Q)
          THEN
            GVL_MSG_AXIS.MetricMessageCtrl.Cmd:= E_MESSAGE_CTRL.MSG_CTRL_WRITE;
          END_IF
        END_IF
    END_CASE

  E_MESSAGE_STATE.MSG_STATE_WRITE:
    CASE eMtrProgress
    OF
      E_PROGRESS.PROGRESS_ERROR,
      E_PROGRESS.PROGRESS_DONE:
        tonIdleWriteMetric(IN := FALSE, PT:= tIdleWriteMetric);
        GVL_MSG_AXIS.MetricMessageCtrl.Cmd    := E_MESSAGE_CTRL.MSG_CTRL_NULL;
    END_CASE
ELSE
    CASE eMtrProgress
    OF
      E_PROGRESS.PROGRESS_DONE:
        GVL_MSG_AXIS.MetricMessageCtrl.Cmd    := E_MESSAGE_CTRL.MSG_CTRL_NULL;
    END_CASE
END_CASE
//-----------------------------------------------------------------------------------------------------------------
//  Metrics/
//-----------------------------------------------------------------------------------------------------------------
//-----------------------------------------------------------------------------------------------------------------

END_PROGRAM

// ---- PLC_MOTION/NCI/NCI.TcPOU
PROGRAM NCI
VAR
  eInit                     : E_PROGRESS;

  nChn,
  nChnInit,
  nAxis,
  nAxisInit                 : UINT;

  stMsg                     : ST_Message;
END_VAR

//-----------------------------------------------------------------------------------------------------------------
// check if compiler define is present [PLC_STATE_DRIVE/CompilerDefines/Manual: NCI]
// see PLC_CONSTANT for conditional pragma
//-----------------------------------------------------------------------------------------------------------------
IF NOT PLC_CONSTANT.NCI_ACTIVE THEN eInit   := E_PROGRESS.PROGRESS_NOT_EXIST; RETURN; END_IF
//-----------------------------------------------------------------------------------------------------------------
//-----------------------------------------------------------------------------------------------------------------
// check for MAIN.eInit
//-----------------------------------------------------------------------------------------------------------------
IF NOT (MAIN_AXIS.eInit = E_PROGRESS.PROGRESS_DONE) THEN eInit   := E_PROGRESS.PROGRESS_INVALID; RETURN; END_IF
//-----------------------------------------------------------------------------------------------------------------
//-----------------------------------------------------------------------------------------------------------------
// /assign dataflow
//-----------------------------------------------------------------------------------------------------------------
FOR nChn := 1 TO MAX_NCI_CH
DO
  // NCI axis configuration --> NC AxisId used
  GVL_NCI.NciCtrl[nChn].ItfChannel.CfgAxes          := ADR(GVL_NCI.AxisConfig[nChn]);

  // R Parameter properties
  GVL_NCI.NciCtrl[nChn].ItfChannel.R_ParameterRead  := ADR(GVL_NCI.R_ParameterRead[nChn]);
  GVL_NCI.NciCtrl[nChn].ItfChannel.R_ParameterWrite := ADR(GVL_NCI.R_ParameterWrite[nChn]);

  // ProgName for channel
  GVL_NCI.NciCtrl[nChn].ItfChannel.Prog             := GVL_NCI.ChannelCtrl[nChn].sProgramName;

  // check REAL value to avoid exception
  IF NOT IsFinite(F_Real(GVL_NCI.ChannelCtrl[nChn].rOverride))
  THEN
    GVL_NCI.NciCtrl[nChn].ItfChannel.Override       := 0.0;
  ELSE
    GVL_NCI.NciCtrl[nChn].ItfChannel.Override       := GVL_NCI.ChannelCtrl[nChn].rOverride;
  END_IF

  // command and state structure assignement
  GVL_NCI.NciCtrl[nChn].ChnCtrl                     := ADR(GVL_NCI.ChannelCtrl[nChn]);
  GVL_NCI.NciCtrl[nChn].ChnState                    := ADR(GVL_NCI.ChannelState[nChn]);
END_FOR
//-----------------------------------------------------------------------------------------------------------------
// assign dataflow/
//-----------------------------------------------------------------------------------------------------------------
//-----------------------------------------------------------------------------------------------------------------
// /INIT
//-----------------------------------------------------------------------------------------------------------------
CASE eInit
OF
  E_PROGRESS.PROGRESS_INVALID:
    FOR nChn := 1 TO MAX_NCI_CH
    DO
      GVL_MSG_AXIS.MessageLevelNciChn[nChn]         := E_MessageType.eMessageVerbose;//GVL_MSG.MessageLevel;
    END_FOR
    nChnInit                                        := 1;
    eInit                                           := E_PROGRESS.PROGRESS_INIT;
  //-----------------------------------------------------------------------------
  //-----------------------------------------------------------------------------
  E_PROGRESS.PROGRESS_INIT:
    stMsg.eType                                     := E_MessageType.eMessageInfo;
    stMsg.eDevice                                   := e_Device.Device_Nci;
    stMsg.eSubdevice                                := e_SubDevice.MainInit;
    stMsg.iErrorNumber                              := MAX_AXIS;
    stMsg.sText                                     := concat('NCI.eInit: ', TO_STRING(eInit));
    f_MessageSet(stMsg);                          

    eInit                                           := E_PROGRESS.PROGRESS_BUSY;
  //-----------------------------------------------------------------------------
  //-----------------------------------------------------------------------------
  E_PROGRESS.PROGRESS_BUSY:
    eInit                                           := E_PROGRESS.PROGRESS_PREPARE;
  //-----------------------------------------------------------------------------
  //-----------------------------------------------------------------------------
  E_PROGRESS.PROGRESS_PREPARE:
    stMsg.eType                                     := E_MessageType.eMessageVerbose;
    stMsg.eDevice                                   := e_Device.Device_Nci;
    stMsg.eSubdevice                                := e_SubDevice.NciStartUp;
    stMsg.iErrorNumber                              := nChnInit;
    stMsg.sText                                     := concat('nChnInit: ', TO_STRING(nChnInit));

    IF (GVL_MSG_AXIS.MessageLevelNciChn[nChnInit] = E_MessageType.eMessageVerbose)
    THEN
      f_MessageSet(stMsg);
    END_IF

    GVL_NCI.ChannelCtrl[nChnInit].eCmd              := E_NCI_CTRL.NULL;
    eInit                                           := E_PROGRESS.PROGRESS_STARTUP;
  //-----------------------------------------------------------------------------
  //-----------------------------------------------------------------------------
  E_PROGRESS.PROGRESS_STARTUP:
    GVL_NCI.ChannelCtrl[nChnInit].eCmd              := E_NCI_CTRL.INIT;

    IF (GVL_NCI.ChannelState[nChnInit].eState = E_NCI_STATE.INIT + E_PROGRESS.PROGRESS_ERROR)
    THEN
      eInit                                         := E_PROGRESS.PROGRESS_ERROR;

      stMsg.eType                                   := E_MessageType.eMessageError;
      stMsg.eDevice                                 := e_Device.Device_Nci;
      stMsg.eSubdevice                              := e_SubDevice.NciStartUp;
      stMsg.iErrorNumber                            := nChnInit;
      stMsg.sText                                   := concat('NCI.eInit ERROR at Index: ', TO_STRING(nChnInit));
      f_MessageSet(stMsg);

    ELSIF (GVL_NCI.ChannelState[nChnInit].eState = E_NCI_STATE.INIT + E_PROGRESS.PROGRESS_DONE)
    THEN
      eInit                                         := E_PROGRESS.PROGRESS_CHECK;
    END_IF
  //-----------------------------------------------------------------------------
  //-----------------------------------------------------------------------------
  E_PROGRESS.PROGRESS_CHECK:
    IF (nChnInit > PLC_CONSTANT.MAX_NCI_CH-1)
    THEN
      eInit                                         := E_PROGRESS.PROGRESS_DONE;

      stMsg.eType                                   := E_MessageType.eMessageInfo;
      stMsg.eDevice                                 := e_Device.Device_Nci;
      stMsg.eSubdevice                              := e_SubDevice.NciStartUp;
      stMsg.iErrorNumber                            := MAX_NCI_CH;
      stMsg.sText                                   := concat('NCI.eInit: ', TO_STRING(eInit));
      f_MessageSet(stMsg);

      FOR nChn := 1 TO MAX_NCI_CH
      DO
        GVL_MSG_AXIS.MessageLevelNciChn[nChn]       := GVL_MSG_AXIS.MessageLevel;
      END_FOR

    ELSE
      nChnInit                                      := nChnInit + 1;
      eInit                                         := E_PROGRESS.PROGRESS_PREPARE;
    END_IF
END_CASE
//-----------------------------------------------------------------------------------------------------------------
// INIT/
//-----------------------------------------------------------------------------------------------------------------
//-----------------------------------------------------------------------------------------------------------------
//-----------------------------------------------------------------------------------------------------------------
// /CYCLE
//-----------------------------------------------------------------------------------------------------------------
FOR nChn := 1 TO MAX_NCI_CH
DO
  // call nci channel controller
  GVL_NCI.NciCtrl[nChn].Cycle();

  GVL_NCI.ProgramNameActive[nChn]                   := GVL_NCI.NciCtrl[nChn].ItfChannel.GetLoadedProg();
  GVL_NCI.ChannelState[nChn].sProgramNameActive     := GVL_NCI.ProgramNameActive[nChn];
  GVL_NCI.NciCtrl[nChn].M_FunctionScope             := ADR(GVL_NCI.M_FunctionCyclic[nChn]);
END_FOR
//-----------------------------------------------------------------------------------------------------------------
// CYCLE/
//-----------------------------------------------------------------------------------------------------------------
//-----------------------------------------------------------------------------------------------------------------

END_PROGRAM

// ---- PLC_MOTION/CAM/CAM.TcPOU
PROGRAM CAM
VAR
  eInit                     : E_PROGRESS;

  nAxis,
  nAxisInit                 : UINT;

  stMsg                     : ST_Message;
END_VAR

//-----------------------------------------------------------------------------------------------------------------
// check if compiler define is present [PLC_MOTION/CompilerDefines/Manual: CAM]
// see PLC_CONSTANT for conditional pragma
//-----------------------------------------------------------------------------------------------------------------
IF NOT PLC_CONSTANT.CAM_ACTIVE THEN eInit := E_PROGRESS.PROGRESS_NOT_EXIST; RETURN; END_IF
//-----------------------------------------------------------------------------------------------------------------
//-----------------------------------------------------------------------------------------------------------------
// check for MAIN.eInit
//-----------------------------------------------------------------------------------------------------------------
IF NOT (MAIN_AXIS.eInit = E_PROGRESS.PROGRESS_DONE) THEN eInit   := E_PROGRESS.PROGRESS_INVALID; RETURN; END_IF
//-----------------------------------------------------------------------------------------------------------------
//-----------------------------------------------------------------------------------------------------------------
// /assign dataflow
//-----------------------------------------------------------------------------------------------------------------
FOR nAxis := 1 TO PLC_CONSTANT.MAX_AXIS
DO
  GVL_CAM.Control[nAxis].ItfMcAxes            := GVL_AXIS.ItfMcAxis;

  GVL_CAM.Control[nAxis].AxisIndex            := nAxis;

  GVL_CAM.Control[nAxis].AxisCtrl             := ADR(GVL_CAM.Ctrl);          // command
  GVL_CAM.Control[nAxis].AxisState            := ADR(GVL_CAM.State);         // state + result of command

  GVL_CAM.Control[nAxis].Axes                 REF=   GVL_AXIS.AxisRef;        // All for one; coupling requires access across all axes

  GVL_CAM.Control[nAxis].AxisInfo             := ADR(GVL_CAM.Info);
  GVL_CAM.Control[nAxis].GearData             := ADR(GVL_CAM.Data);

